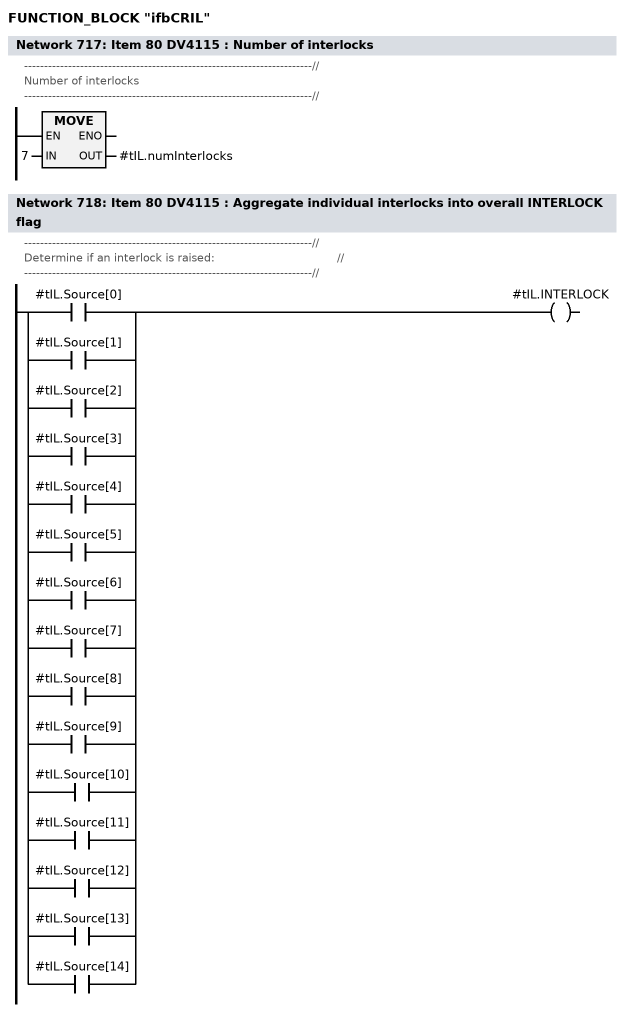
    L 7;
    T #tIL.numInterlocks;

NETWORK
TITLE = Item 80 DV4115 : Aggregate individual interlocks into overall INTERLOCK flag
    //------------------------------------------------------------------------//
    // Determine if an interlock is raised:                                   //
    //------------------------------------------------------------------------//
    O #tIL.Source[0];
    O #tIL.Source[1];
    O #tIL.Source[2];
    O #tIL.Source[3];
    O #tIL.Source[4];
    O #tIL.Source[5];
    O #tIL.Source[6];
    O #tIL.Source[7];
    O #tIL.Source[8];
    O #tIL.Source[9];
    O #tIL.Source[10];
    O #tIL.Source[11];
    O #tIL.Source[12];
    O #tIL.Source[13];
    O #tIL.Source[14];
    = #tIL.INTERLOCK;

NETWORK
TITLE = Item 80 DV4115 : Update the instance data
    //------------------------------------------------------------------------//
    // Update the instance DB with the calculated interlock flags:            //
    //------------------------------------------------------------------------//
    CALL MOVE
    {value_type := 'Variant'}
    (   IN                   := #tIL ,
        OUT                  := #p[80]
    );

NETWORK
TITLE = Item 81 DV4117 : Spray Ball 1 Valve initialise variables
    //------------------------------------------------------------------------//
    // CRITICAL INTERLOCK   CRITICAL INTERLOCK   CRITICAL INTERLOCK   CRITICA //
    // CRITICAL INTERLOCK   CRITICAL INTERLOCK   CRITICAL INTERLOCK   CRITICA //
    //                                                                        //
    // Clear the interlock flag:                                              //
    //------------------------------------------------------------------------//
    A "alwaysLow";
    = #tIL.INTERLOCK;

    //------------------------------------------------------------------------//
    // Clear all interlock values to initialise them to off:                  //
    //------------------------------------------------------------------------//
    CALL FILL_BLK
    {value_type := 'Bool', count_type := 'UInt'}
    (   IN                   := 0 ,
        COUNT                := 15 ,
        OUT                  := #tIL.Source[0]
    );


NETWORK
TITLE = Item 81 DV4117 interlock source : A RD4101 Vessel Burst Disc ALARM
    //------------------------------------------------------------------------//
    // Calculate the interlock condition:                                     //
    //------------------------------------------------------------------------//
    A idbDI1.f[16].p.read.mc.INTERLOCK;
    = #tIL.Source[0];

NETWORK
TITLE = Item 81 DV4117 interlock source : A ES4100 Vessel Emergency Stop mounted on HMI INTERLOCK
    //------------------------------------------------------------------------//
    // Calculate the interlock condition:                                     //
    //------------------------------------------------------------------------//
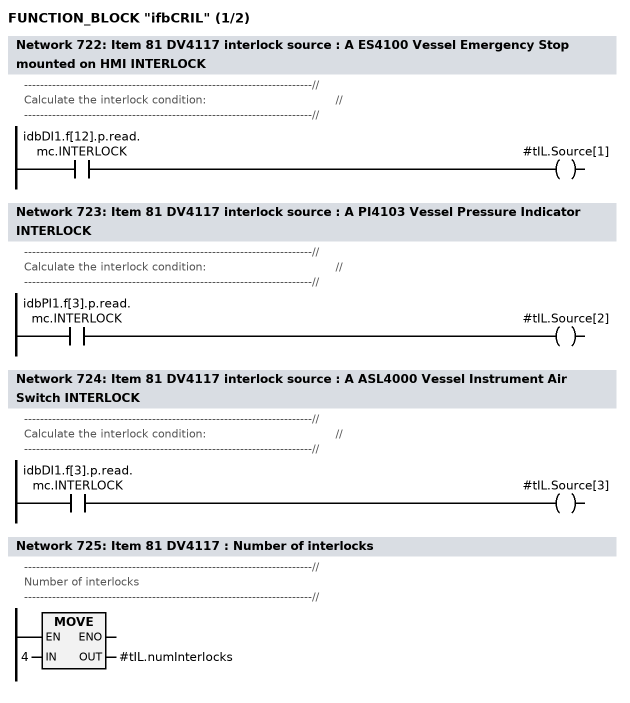
    A idbDI1.f[12].p.read.mc.INTERLOCK;
    = #tIL.Source[1];

NETWORK
TITLE = Item 81 DV4117 interlock source : A PI4103 Vessel Pressure Indicator INTERLOCK
    //------------------------------------------------------------------------//
    // Calculate the interlock condition:                                     //
    //------------------------------------------------------------------------//
    A idbPI1.f[3].p.read.mc.INTERLOCK;
    = #tIL.Source[2];

NETWORK
TITLE = Item 81 DV4117 interlock source : A ASL4000 Vessel Instrument Air Switch INTERLOCK
    //------------------------------------------------------------------------//
    // Calculate the interlock condition:                                     //
    //------------------------------------------------------------------------//
    A idbDI1.f[3].p.read.mc.INTERLOCK;
    = #tIL.Source[3];


NETWORK
TITLE = Item 81 DV4117 : Number of interlocks
    //------------------------------------------------------------------------//
    // Number of interlocks
    //------------------------------------------------------------------------//
    L 4;
    T #tIL.numInterlocks;

NETWORK
TITLE = Item 81 DV4117 : Aggregate individual interlocks into overall INTERLOCK flag
    //------------------------------------------------------------------------//
    // Determine if an interlock is raised:                                   //
    //------------------------------------------------------------------------//
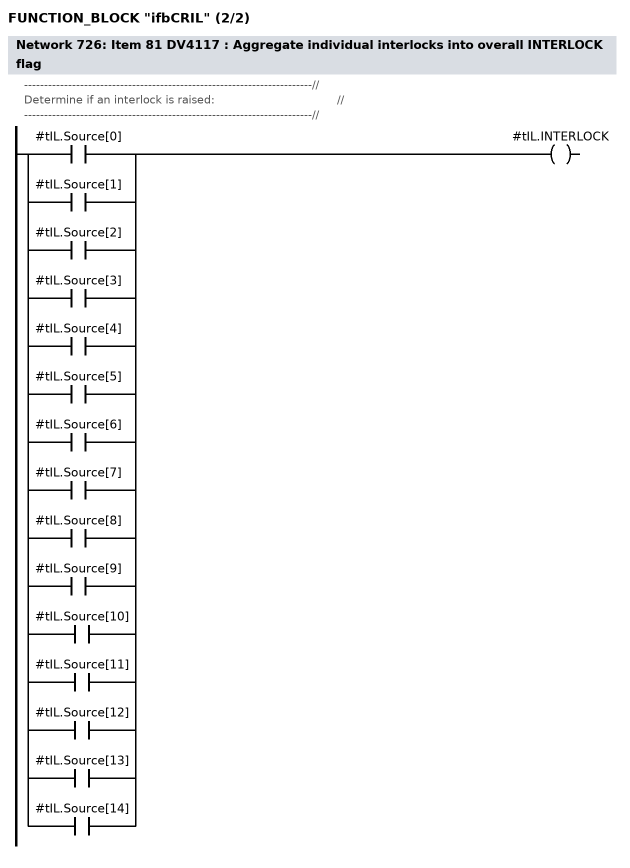
    O #tIL.Source[0];
    O #tIL.Source[1];
    O #tIL.Source[2];
    O #tIL.Source[3];
    O #tIL.Source[4];
    O #tIL.Source[5];
    O #tIL.Source[6];
    O #tIL.Source[7];
    O #tIL.Source[8];
    O #tIL.Source[9];
    O #tIL.Source[10];
    O #tIL.Source[11];
    O #tIL.Source[12];
    O #tIL.Source[13];
    O #tIL.Source[14];
    = #tIL.INTERLOCK;

NETWORK
TITLE = Item 81 DV4117 : Update the instance data
    //------------------------------------------------------------------------//
    // Update the instance DB with the calculated interlock flags:            //
    //------------------------------------------------------------------------//
    CALL MOVE
    {value_type := 'Variant'}
    (   IN                   := #tIL ,
        OUT                  := #p[81]
    );

NETWORK
TITLE = Item 82 DV4119 : Spray Ball 2 Valve initialise variables
    //------------------------------------------------------------------------//
    // CRITICAL INTERLOCK   CRITICAL INTERLOCK   CRITICAL INTERLOCK   CRITICA //
    // CRITICAL INTERLOCK   CRITICAL INTERLOCK   CRITICAL INTERLOCK   CRITICA //
    //                                                                        //
    // Clear the interlock flag:                                              //
    //------------------------------------------------------------------------//
    A "alwaysLow";
    = #tIL.INTERLOCK;

    //------------------------------------------------------------------------//
    // Clear all interlock values to initialise them to off:                  //
    //------------------------------------------------------------------------//
    CALL FILL_BLK
    {value_type := 'Bool', count_type := 'UInt'}
    (   IN                   := 0 ,
        COUNT                := 15 ,
        OUT                  := #tIL.Source[0]
    );


NETWORK
TITLE = Item 82 DV4119 interlock source : A RD4101 Vessel Burst Disc ALARM
    //------------------------------------------------------------------------//
    // Calculate the interlock condition:                                     //
    //------------------------------------------------------------------------//
    A idbDI1.f[16].p.read.mc.INTERLOCK;
    = #tIL.Source[0];

NETWORK
TITLE = Item 82 DV4119 interlock source : A ES4100 Vessel Emergency Stop mounted on HMI INTERLOCK
    //------------------------------------------------------------------------//
    // Calculate the interlock condition:                                     //
    //------------------------------------------------------------------------//
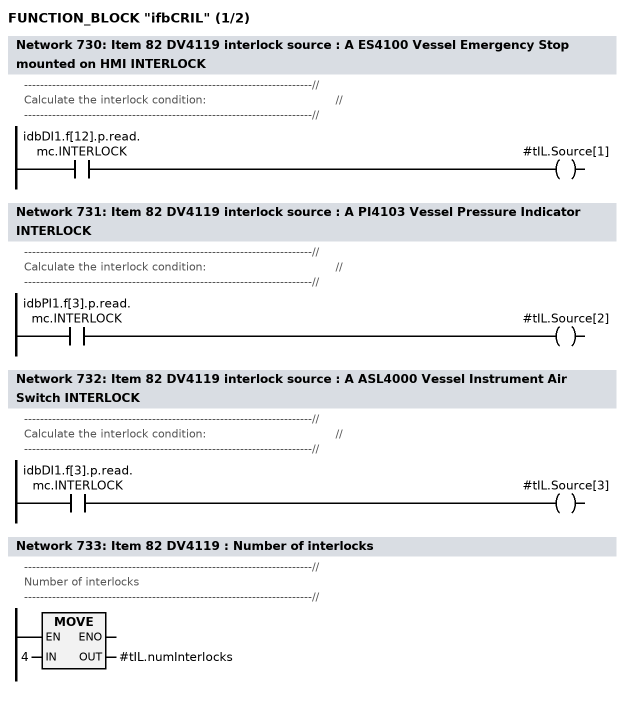
    A idbDI1.f[12].p.read.mc.INTERLOCK;
    = #tIL.Source[1];

NETWORK
TITLE = Item 82 DV4119 interlock source : A PI4103 Vessel Pressure Indicator INTERLOCK
    //------------------------------------------------------------------------//
    // Calculate the interlock condition:                                     //
    //------------------------------------------------------------------------//
    A idbPI1.f[3].p.read.mc.INTERLOCK;
    = #tIL.Source[2];

NETWORK
TITLE = Item 82 DV4119 interlock source : A ASL4000 Vessel Instrument Air Switch INTERLOCK
    //------------------------------------------------------------------------//
    // Calculate the interlock condition:                                     //
    //------------------------------------------------------------------------//
    A idbDI1.f[3].p.read.mc.INTERLOCK;
    = #tIL.Source[3];


NETWORK
TITLE = Item 82 DV4119 : Number of interlocks
    //------------------------------------------------------------------------//
    // Number of interlocks
    //------------------------------------------------------------------------//
    L 4;
    T #tIL.numInterlocks;

NETWORK
TITLE = Item 82 DV4119 : Aggregate individual interlocks into overall INTERLOCK flag
    //------------------------------------------------------------------------//
    // Determine if an interlock is raised:                                   //
    //------------------------------------------------------------------------//
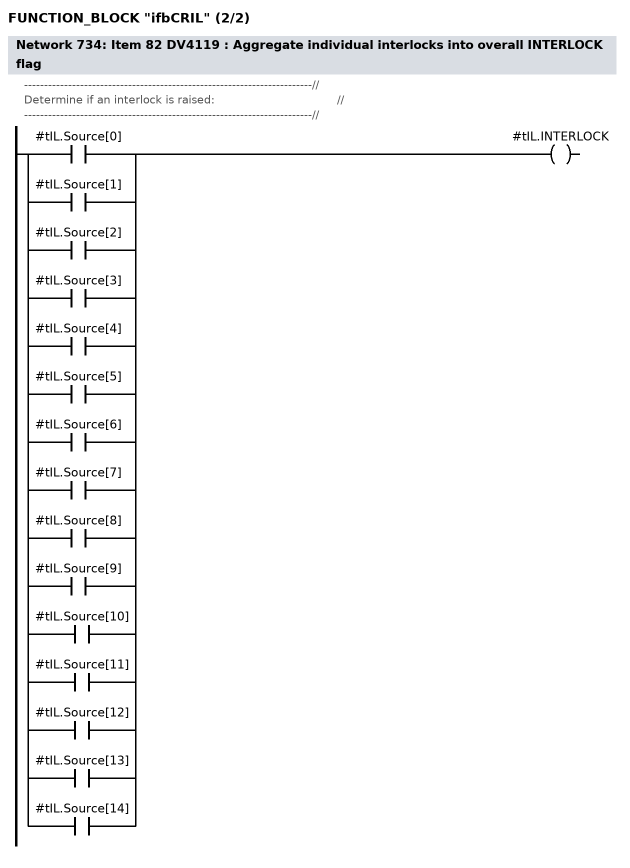
    O #tIL.Source[0];
    O #tIL.Source[1];
    O #tIL.Source[2];
    O #tIL.Source[3];
    O #tIL.Source[4];
    O #tIL.Source[5];
    O #tIL.Source[6];
    O #tIL.Source[7];
    O #tIL.Source[8];
    O #tIL.Source[9];
    O #tIL.Source[10];
    O #tIL.Source[11];
    O #tIL.Source[12];
    O #tIL.Source[13];
    O #tIL.Source[14];
    = #tIL.INTERLOCK;

NETWORK
TITLE = Item 82 DV4119 : Update the instance data
    //------------------------------------------------------------------------//
    // Update the instance DB with the calculated interlock flags:            //
    //------------------------------------------------------------------------//
    CALL MOVE
    {value_type := 'Variant'}
    (   IN                   := #tIL ,
        OUT                  := #p[82]
    );

NETWORK
TITLE = Item 83 DV4121 : Outlet Valve initialise variables
    //------------------------------------------------------------------------//
    // CRITICAL INTERLOCK   CRITICAL INTERLOCK   CRITICAL INTERLOCK   CRITICA //
    // CRITICAL INTERLOCK   CRITICAL INTERLOCK   CRITICAL INTERLOCK   CRITICA //
    //                                                                        //
    // Clear the interlock flag:                                              //
    //------------------------------------------------------------------------//
    A "alwaysLow";
    = #tIL.INTERLOCK;

    //------------------------------------------------------------------------//
    // Clear all interlock values to initialise them to off:                  //
    //------------------------------------------------------------------------//
    CALL FILL_BLK
    {value_type := 'Bool', count_type := 'UInt'}
    (   IN                   := 0 ,
        COUNT                := 15 ,
        OUT                  := #tIL.Source[0]
    );


NETWORK
TITLE = Item 83 DV4121 interlock source : A RD4101 Vessel Burst Disc ALARM
    //------------------------------------------------------------------------//
    // Calculate the interlock condition:                                     //
    //------------------------------------------------------------------------//
    A idbDI1.f[16].p.read.mc.INTERLOCK;
    = #tIL.Source[0];

NETWORK
TITLE = Item 83 DV4121 interlock source : A ES4100 Vessel Emergency Stop mounted on HMI INTERLOCK
    //------------------------------------------------------------------------//
    // Calculate the interlock condition:                                     //
    //------------------------------------------------------------------------//
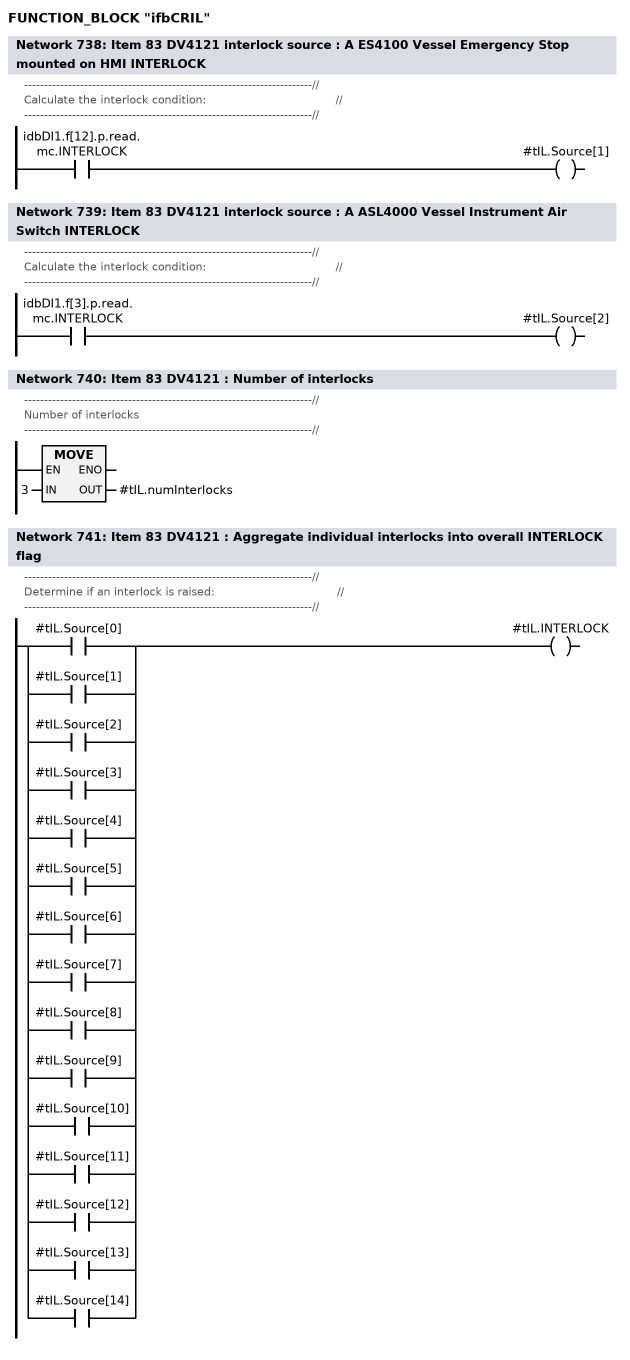
    A idbDI1.f[12].p.read.mc.INTERLOCK;
    = #tIL.Source[1];

NETWORK
TITLE = Item 83 DV4121 interlock source : A ASL4000 Vessel Instrument Air Switch INTERLOCK
    //------------------------------------------------------------------------//
    // Calculate the interlock condition:                                     //
    //------------------------------------------------------------------------//
    A idbDI1.f[3].p.read.mc.INTERLOCK;
    = #tIL.Source[2];


NETWORK
TITLE = Item 83 DV4121 : Number of interlocks
    //------------------------------------------------------------------------//
    // Number of interlocks
    //------------------------------------------------------------------------//
    L 3;
    T #tIL.numInterlocks;

NETWORK
TITLE = Item 83 DV4121 : Aggregate individual interlocks into overall INTERLOCK flag
    //------------------------------------------------------------------------//
    // Determine if an interlock is raised:                                   //
    //------------------------------------------------------------------------//
    O #tIL.Source[0];
    O #tIL.Source[1];
    O #tIL.Source[2];
    O #tIL.Source[3];
    O #tIL.Source[4];
    O #tIL.Source[5];
    O #tIL.Source[6];
    O #tIL.Source[7];
    O #tIL.Source[8];
    O #tIL.Source[9];
    O #tIL.Source[10];
    O #tIL.Source[11];
    O #tIL.Source[12];
    O #tIL.Source[13];
    O #tIL.Source[14];
    = #tIL.INTERLOCK;

NETWORK
TITLE = Item 83 DV4121 : Update the instance data
    //------------------------------------------------------------------------//
    // Update the instance DB with the calculated interlock flags:            //
    //------------------------------------------------------------------------//
    CALL MOVE
    {value_type := 'Variant'}
    (   IN                   := #tIL ,
        OUT                  := #p[83]
    );

NETWORK
TITLE = Item 84 DV4125 : Sy Transfer line Valve Matrix SMFLx initialise variables
    //------------------------------------------------------------------------//
    // CRITICAL INTERLOCK   CRITICAL INTERLOCK   CRITICAL INTERLOCK   CRITICA //
    // CRITICAL INTERLOCK   CRITICAL INTERLOCK   CRITICAL INTERLOCK   CRITICA //
    //                                                                        //
    // Clear the interlock flag:                                              //
    //------------------------------------------------------------------------//
    A "alwaysLow";
    = #tIL.INTERLOCK;

    //------------------------------------------------------------------------//
    // Clear all interlock values to initialise them to off:                  //
    //------------------------------------------------------------------------//
    CALL FILL_BLK
    {value_type := 'Bool', count_type := 'UInt'}
    (   IN                   := 0 ,
        COUNT                := 15 ,
        OUT                  := #tIL.Source[0]
    );


NETWORK
TITLE = Item 84 DV4125 interlock source : AN ZSC4111 SMFL1 to S1/BFS1 Flowpath Indicator IN   AN ZSC4113 SMFL2 to S1/BFS1 Flowpath Indicator IN
    //------------------------------------------------------------------------//
    // Calculate the interlock condition:                                     //
    //------------------------------------------------------------------------//
    AN(;
    L "idbZSC2".f[24].p.read.mc.STATE;
    L "dbCONST".BLK.ZSC2.STATE.IN;
    ==I;
    );
AN(;
    L "idbZSC2".f[25].p.read.mc.STATE;
    L "dbCONST".BLK.ZSC2.STATE.IN;
    ==I;
    );
    = #tIL.Source[0];


NETWORK
TITLE = Item 84 DV4125 : Number of interlocks
    //------------------------------------------------------------------------//
    // Number of interlocks
    //------------------------------------------------------------------------//
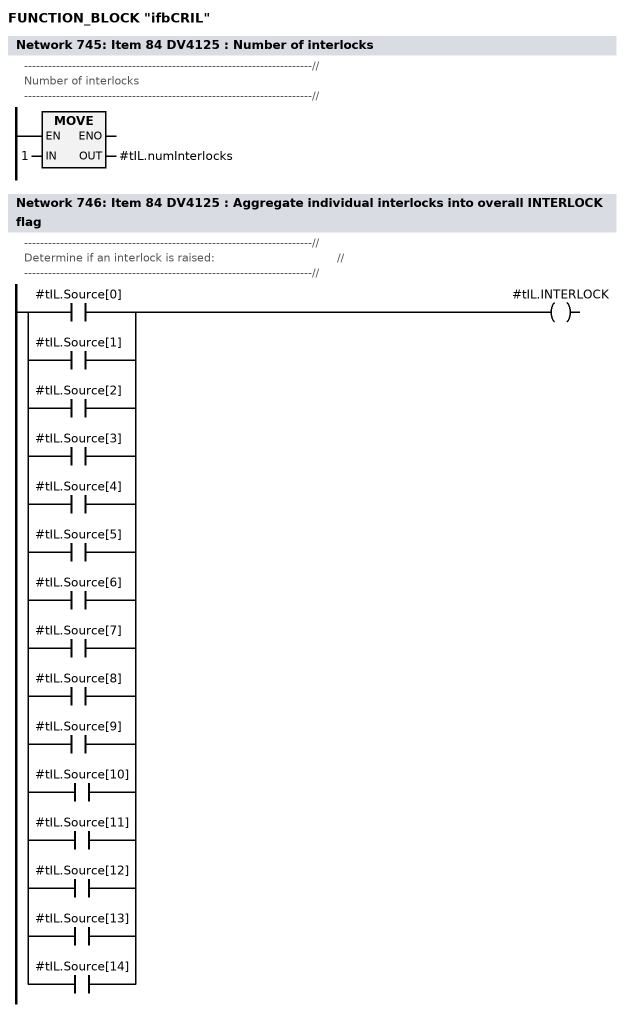
    L 1;
    T #tIL.numInterlocks;

NETWORK
TITLE = Item 84 DV4125 : Aggregate individual interlocks into overall INTERLOCK flag
    //------------------------------------------------------------------------//
    // Determine if an interlock is raised:                                   //
    //------------------------------------------------------------------------//
    O #tIL.Source[0];
    O #tIL.Source[1];
    O #tIL.Source[2];
    O #tIL.Source[3];
    O #tIL.Source[4];
    O #tIL.Source[5];
    O #tIL.Source[6];
    O #tIL.Source[7];
    O #tIL.Source[8];
    O #tIL.Source[9];
    O #tIL.Source[10];
    O #tIL.Source[11];
    O #tIL.Source[12];
    O #tIL.Source[13];
    O #tIL.Source[14];
    = #tIL.INTERLOCK;

NETWORK
TITLE = Item 84 DV4125 : Update the instance data
    //------------------------------------------------------------------------//
    // Update the instance DB with the calculated interlock flags:            //
    //------------------------------------------------------------------------//
    CALL MOVE
    {value_type := 'Variant'}
    (   IN                   := #tIL ,
        OUT                  := #p[84]
    );

NETWORK
TITLE = Item 85 DV4129 : Sy Transfer line Valve Matrix FLz initialise variables
    //------------------------------------------------------------------------//
    // CRITICAL INTERLOCK   CRITICAL INTERLOCK   CRITICAL INTERLOCK   CRITICA //
    // CRITICAL INTERLOCK   CRITICAL INTERLOCK   CRITICAL INTERLOCK   CRITICA //
    //                                                                        //
    // Clear the interlock flag:                                              //
    //------------------------------------------------------------------------//
    A "alwaysLow";
    = #tIL.INTERLOCK;

    //------------------------------------------------------------------------//
    // Clear all interlock values to initialise them to off:                  //
    //------------------------------------------------------------------------//
    CALL FILL_BLK
    {value_type := 'Bool', count_type := 'UInt'}
    (   IN                   := 0 ,
        COUNT                := 15 ,
        OUT                  := #tIL.Source[0]
    );


NETWORK
TITLE = Item 85 DV4129 interlock source : AN ZSC4115 S1 to F1P1 Flowpath Indicator IN   AN ZSC4117 S1 to F2P1 Flowpath Indicator IN
    //------------------------------------------------------------------------//
    // Calculate the interlock condition:                                     //
    //------------------------------------------------------------------------//
    AN(;
    L "idbZSC2".f[26].p.read.mc.STATE;
    L "dbCONST".BLK.ZSC2.STATE.IN;
    ==I;
    );
AN(;
    L "idbZSC2".f[27].p.read.mc.STATE;
    L "dbCONST".BLK.ZSC2.STATE.IN;
    ==I;
    );
    = #tIL.Source[0];


NETWORK
TITLE = Item 85 DV4129 : Number of interlocks
    //------------------------------------------------------------------------//
    // Number of interlocks
    //------------------------------------------------------------------------//
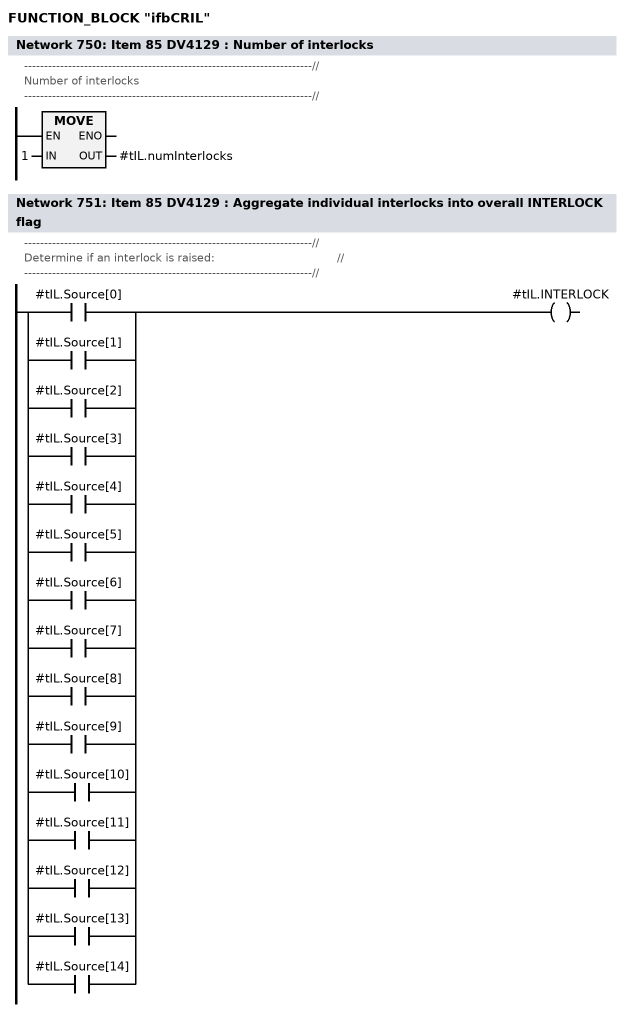
    L 1;
    T #tIL.numInterlocks;

NETWORK
TITLE = Item 85 DV4129 : Aggregate individual interlocks into overall INTERLOCK flag
    //------------------------------------------------------------------------//
    // Determine if an interlock is raised:                                   //
    //------------------------------------------------------------------------//
    O #tIL.Source[0];
    O #tIL.Source[1];
    O #tIL.Source[2];
    O #tIL.Source[3];
    O #tIL.Source[4];
    O #tIL.Source[5];
    O #tIL.Source[6];
    O #tIL.Source[7];
    O #tIL.Source[8];
    O #tIL.Source[9];
    O #tIL.Source[10];
    O #tIL.Source[11];
    O #tIL.Source[12];
    O #tIL.Source[13];
    O #tIL.Source[14];
    = #tIL.INTERLOCK;

NETWORK
TITLE = Item 85 DV4129 : Update the instance data
    //------------------------------------------------------------------------//
    // Update the instance DB with the calculated interlock flags:            //
    //------------------------------------------------------------------------//
    CALL MOVE
    {value_type := 'Variant'}
    (   IN                   := #tIL ,
        OUT                  := #p[85]
    );

NETWORK
TITLE = Item 86 HE1101 : Electric Heating Element initialise variables
    //------------------------------------------------------------------------//
    // CRITICAL INTERLOCK   CRITICAL INTERLOCK   CRITICAL INTERLOCK   CRITICA //
    // CRITICAL INTERLOCK   CRITICAL INTERLOCK   CRITICAL INTERLOCK   CRITICA //
    //                                                                        //
    // Clear the interlock flag:                                              //
    //------------------------------------------------------------------------//
    A "alwaysLow";
    = #tIL.INTERLOCK;

    //------------------------------------------------------------------------//
    // Clear all interlock values to initialise them to off:                  //
    //------------------------------------------------------------------------//
    CALL FILL_BLK
    {value_type := 'Bool', count_type := 'UInt'}
    (   IN                   := 0 ,
        COUNT                := 15 ,
        OUT                  := #tIL.Source[0]
    );


NETWORK
TITLE = Item 86 HE1101 interlock source : A RD1101 Vessel Burst Disc ALARM
    //------------------------------------------------------------------------//
    // Calculate the interlock condition:                                     //
    //------------------------------------------------------------------------//
    A idbDI1.f[13].p.read.mc.INTERLOCK;
    = #tIL.Source[0];

NETWORK
TITLE = Item 86 HE1101 interlock source : A ES1100 Vessel Emergency Stop mounted on HMI INTERLOCK
    //------------------------------------------------------------------------//
    // Calculate the interlock condition:                                     //
    //------------------------------------------------------------------------//
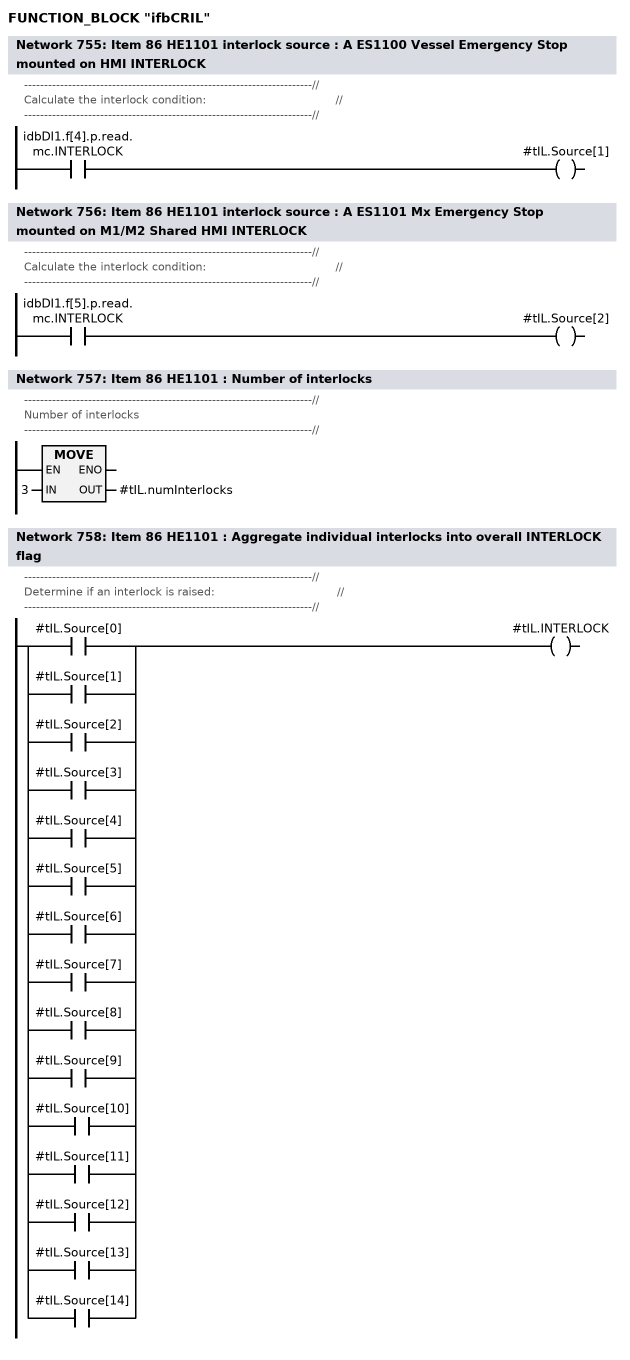
    A idbDI1.f[4].p.read.mc.INTERLOCK;
    = #tIL.Source[1];

NETWORK
TITLE = Item 86 HE1101 interlock source : A ES1101 Mx Emergency Stop mounted on M1/M2 Shared HMI INTERLOCK
    //------------------------------------------------------------------------//
    // Calculate the interlock condition:                                     //
    //------------------------------------------------------------------------//
    A idbDI1.f[5].p.read.mc.INTERLOCK;
    = #tIL.Source[2];


NETWORK
TITLE = Item 86 HE1101 : Number of interlocks
    //------------------------------------------------------------------------//
    // Number of interlocks
    //------------------------------------------------------------------------//
    L 3;
    T #tIL.numInterlocks;

NETWORK
TITLE = Item 86 HE1101 : Aggregate individual interlocks into overall INTERLOCK flag
    //------------------------------------------------------------------------//
    // Determine if an interlock is raised:                                   //
    //------------------------------------------------------------------------//
    O #tIL.Source[0];
    O #tIL.Source[1];
    O #tIL.Source[2];
    O #tIL.Source[3];
    O #tIL.Source[4];
    O #tIL.Source[5];
    O #tIL.Source[6];
    O #tIL.Source[7];
    O #tIL.Source[8];
    O #tIL.Source[9];
    O #tIL.Source[10];
    O #tIL.Source[11];
    O #tIL.Source[12];
    O #tIL.Source[13];
    O #tIL.Source[14];
    = #tIL.INTERLOCK;

NETWORK
TITLE = Item 86 HE1101 : Update the instance data
    //------------------------------------------------------------------------//
    // Update the instance DB with the calculated interlock flags:            //
    //------------------------------------------------------------------------//
    CALL MOVE
    {value_type := 'Variant'}
    (   IN                   := #tIL ,
        OUT                  := #p[86]
    );

NETWORK
TITLE = Item 87 HE2101 : Electric Heating Element initialise variables
    //------------------------------------------------------------------------//
    // CRITICAL INTERLOCK   CRITICAL INTERLOCK   CRITICAL INTERLOCK   CRITICA //
    // CRITICAL INTERLOCK   CRITICAL INTERLOCK   CRITICAL INTERLOCK   CRITICA //
    //                                                                        //
    // Clear the interlock flag:                                              //
    //------------------------------------------------------------------------//
    A "alwaysLow";
    = #tIL.INTERLOCK;

    //------------------------------------------------------------------------//
    // Clear all interlock values to initialise them to off:                  //
    //------------------------------------------------------------------------//
    CALL FILL_BLK
    {value_type := 'Bool', count_type := 'UInt'}
    (   IN                   := 0 ,
        COUNT                := 15 ,
        OUT                  := #tIL.Source[0]
    );


NETWORK
TITLE = Item 87 HE2101 interlock source : A RD2101 Vessel Burst Disc ALARM
    //------------------------------------------------------------------------//
    // Calculate the interlock condition:                                     //
    //------------------------------------------------------------------------//
    A idbDI1.f[14].p.read.mc.INTERLOCK;
    = #tIL.Source[0];

NETWORK
TITLE = Item 87 HE2101 interlock source : A ES2100 Vessel Emergency Stop mounted on HMI INTERLOCK
    //------------------------------------------------------------------------//
    // Calculate the interlock condition:                                     //
    //------------------------------------------------------------------------//
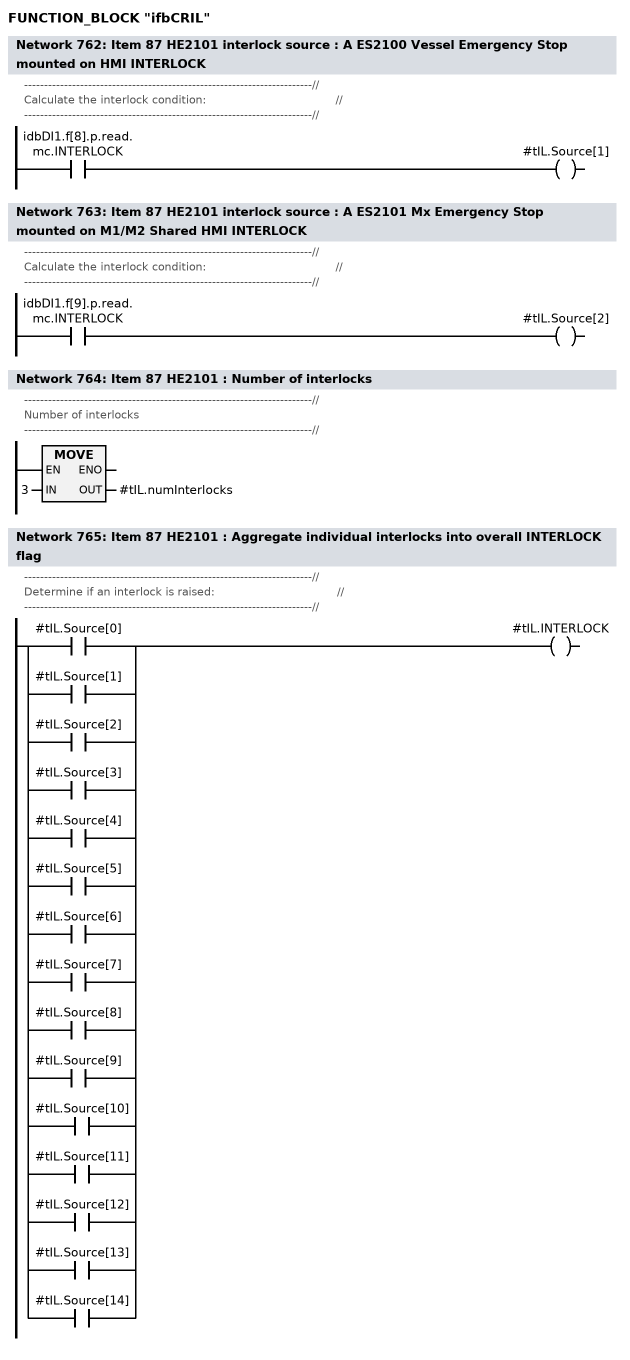
    A idbDI1.f[8].p.read.mc.INTERLOCK;
    = #tIL.Source[1];

NETWORK
TITLE = Item 87 HE2101 interlock source : A ES2101 Mx Emergency Stop mounted on M1/M2 Shared HMI INTERLOCK
    //------------------------------------------------------------------------//
    // Calculate the interlock condition:                                     //
    //------------------------------------------------------------------------//
    A idbDI1.f[9].p.read.mc.INTERLOCK;
    = #tIL.Source[2];


NETWORK
TITLE = Item 87 HE2101 : Number of interlocks
    //------------------------------------------------------------------------//
    // Number of interlocks
    //------------------------------------------------------------------------//
    L 3;
    T #tIL.numInterlocks;

NETWORK
TITLE = Item 87 HE2101 : Aggregate individual interlocks into overall INTERLOCK flag
    //------------------------------------------------------------------------//
    // Determine if an interlock is raised:                                   //
    //------------------------------------------------------------------------//
    O #tIL.Source[0];
    O #tIL.Source[1];
    O #tIL.Source[2];
    O #tIL.Source[3];
    O #tIL.Source[4];
    O #tIL.Source[5];
    O #tIL.Source[6];
    O #tIL.Source[7];
    O #tIL.Source[8];
    O #tIL.Source[9];
    O #tIL.Source[10];
    O #tIL.Source[11];
    O #tIL.Source[12];
    O #tIL.Source[13];
    O #tIL.Source[14];
    = #tIL.INTERLOCK;

NETWORK
TITLE = Item 87 HE2101 : Update the instance data
    //------------------------------------------------------------------------//
    // Update the instance DB with the calculated interlock flags:            //
    //------------------------------------------------------------------------//
    CALL MOVE
    {value_type := 'Variant'}
    (   IN                   := #tIL ,
        OUT                  := #p[87]
    );

NETWORK
TITLE = Item 88 HE3101 : Electric Heating Element initialise variables
    //------------------------------------------------------------------------//
    // CRITICAL INTERLOCK   CRITICAL INTERLOCK   CRITICAL INTERLOCK   CRITICA //
    // CRITICAL INTERLOCK   CRITICAL INTERLOCK   CRITICAL INTERLOCK   CRITICA //
    //                                                                        //
    // Clear the interlock flag:                                              //
    //------------------------------------------------------------------------//
    A "alwaysLow";
    = #tIL.INTERLOCK;

    //------------------------------------------------------------------------//
    // Clear all interlock values to initialise them to off:                  //
    //------------------------------------------------------------------------//
    CALL FILL_BLK
    {value_type := 'Bool', count_type := 'UInt'}
    (   IN                   := 0 ,
        COUNT                := 15 ,
        OUT                  := #tIL.Source[0]
    );


NETWORK
TITLE = Item 88 HE3101 interlock source : A RD3101 Vessel Burst Disc ALARM
    //------------------------------------------------------------------------//
    // Calculate the interlock condition:                                     //
    //------------------------------------------------------------------------//
    A idbDI1.f[15].p.read.mc.INTERLOCK;
    = #tIL.Source[0];

NETWORK
TITLE = Item 88 HE3101 interlock source : A ES3100 Vessel Emergency Stop mounted on HMI INTERLOCK
    //------------------------------------------------------------------------//
    // Calculate the interlock condition:                                     //
    //------------------------------------------------------------------------//
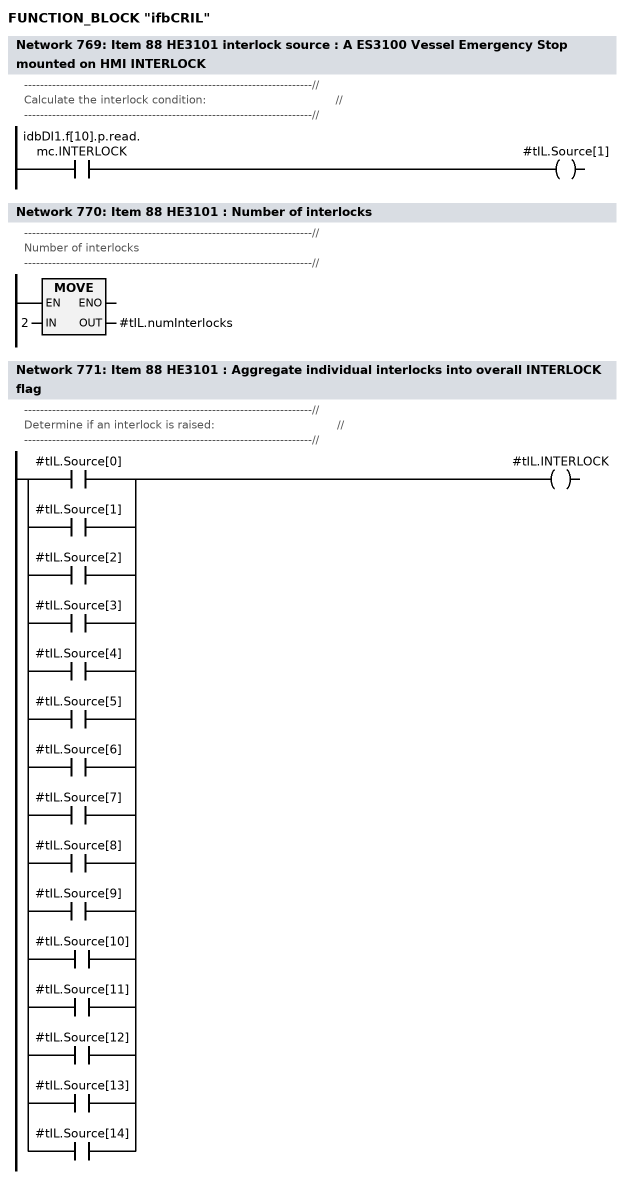
    A idbDI1.f[10].p.read.mc.INTERLOCK;
    = #tIL.Source[1];


NETWORK
TITLE = Item 88 HE3101 : Number of interlocks
    //------------------------------------------------------------------------//
    // Number of interlocks
    //------------------------------------------------------------------------//
    L 2;
    T #tIL.numInterlocks;

NETWORK
TITLE = Item 88 HE3101 : Aggregate individual interlocks into overall INTERLOCK flag
    //------------------------------------------------------------------------//
    // Determine if an interlock is raised:                                   //
    //------------------------------------------------------------------------//
    O #tIL.Source[0];
    O #tIL.Source[1];
    O #tIL.Source[2];
    O #tIL.Source[3];
    O #tIL.Source[4];
    O #tIL.Source[5];
    O #tIL.Source[6];
    O #tIL.Source[7];
    O #tIL.Source[8];
    O #tIL.Source[9];
    O #tIL.Source[10];
    O #tIL.Source[11];
    O #tIL.Source[12];
    O #tIL.Source[13];
    O #tIL.Source[14];
    = #tIL.INTERLOCK;

NETWORK
TITLE = Item 88 HE3101 : Update the instance data
    //------------------------------------------------------------------------//
    // Update the instance DB with the calculated interlock flags:            //
    //------------------------------------------------------------------------//
    CALL MOVE
    {value_type := 'Variant'}
    (   IN                   := #tIL ,
        OUT                  := #p[88]
    );

NETWORK
TITLE = Item 89 HE4101 : Electric Heating Element initialise variables
    //------------------------------------------------------------------------//
    // CRITICAL INTERLOCK   CRITICAL INTERLOCK   CRITICAL INTERLOCK   CRITICA //
    // CRITICAL INTERLOCK   CRITICAL INTERLOCK   CRITICAL INTERLOCK   CRITICA //
    //                                                                        //
    // Clear the interlock flag:                                              //
    //------------------------------------------------------------------------//
    A "alwaysLow";
    = #tIL.INTERLOCK;

    //------------------------------------------------------------------------//
    // Clear all interlock values to initialise them to off:                  //
    //------------------------------------------------------------------------//
    CALL FILL_BLK
    {value_type := 'Bool', count_type := 'UInt'}
    (   IN                   := 0 ,
        COUNT                := 15 ,
        OUT                  := #tIL.Source[0]
    );


NETWORK
TITLE = Item 89 HE4101 interlock source : A RD4101 Vessel Burst Disc ALARM
    //------------------------------------------------------------------------//
    // Calculate the interlock condition:                                     //
    //------------------------------------------------------------------------//
    A idbDI1.f[16].p.read.mc.INTERLOCK;
    = #tIL.Source[0];

NETWORK
TITLE = Item 89 HE4101 interlock source : A ES4100 Vessel Emergency Stop mounted on HMI INTERLOCK
    //------------------------------------------------------------------------//
    // Calculate the interlock condition:                                     //
    //------------------------------------------------------------------------//
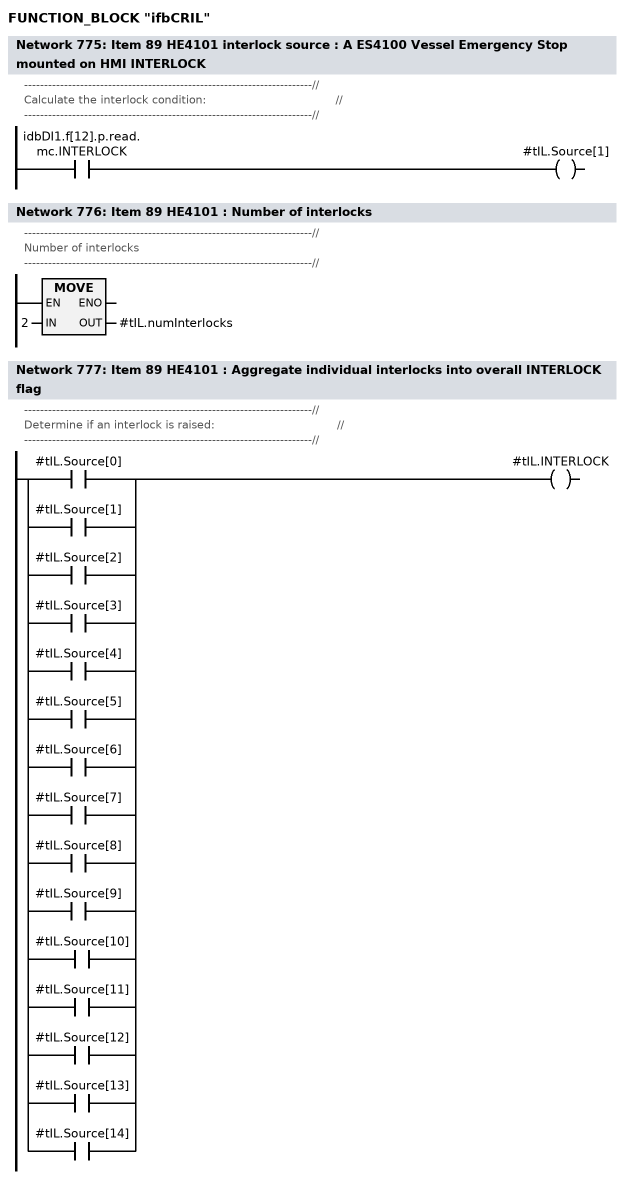
    A idbDI1.f[12].p.read.mc.INTERLOCK;
    = #tIL.Source[1];


NETWORK
TITLE = Item 89 HE4101 : Number of interlocks
    //------------------------------------------------------------------------//
    // Number of interlocks
    //------------------------------------------------------------------------//
    L 2;
    T #tIL.numInterlocks;

NETWORK
TITLE = Item 89 HE4101 : Aggregate individual interlocks into overall INTERLOCK flag
    //------------------------------------------------------------------------//
    // Determine if an interlock is raised:                                   //
    //------------------------------------------------------------------------//
    O #tIL.Source[0];
    O #tIL.Source[1];
    O #tIL.Source[2];
    O #tIL.Source[3];
    O #tIL.Source[4];
    O #tIL.Source[5];
    O #tIL.Source[6];
    O #tIL.Source[7];
    O #tIL.Source[8];
    O #tIL.Source[9];
    O #tIL.Source[10];
    O #tIL.Source[11];
    O #tIL.Source[12];
    O #tIL.Source[13];
    O #tIL.Source[14];
    = #tIL.INTERLOCK;

NETWORK
TITLE = Item 89 HE4101 : Update the instance data
    //------------------------------------------------------------------------//
    // Update the instance DB with the calculated interlock flags:            //
    //------------------------------------------------------------------------//
    CALL MOVE
    {value_type := 'Variant'}
    (   IN                   := #tIL ,
        OUT                  := #p[89]
    );

NETWORK
TITLE = Item 90 PC1103 : Pressure Control initialise variables
    //------------------------------------------------------------------------//
    // CRITICAL INTERLOCK   CRITICAL INTERLOCK   CRITICAL INTERLOCK   CRITICA //
    // CRITICAL INTERLOCK   CRITICAL INTERLOCK   CRITICAL INTERLOCK   CRITICA //
    //                                                                        //
    // Clear the interlock flag:                                              //
    //------------------------------------------------------------------------//
    A "alwaysLow";
    = #tIL.INTERLOCK;

    //------------------------------------------------------------------------//
    // Clear all interlock values to initialise them to off:                  //
    //------------------------------------------------------------------------//
    CALL FILL_BLK
    {value_type := 'Bool', count_type := 'UInt'}
    (   IN                   := 0 ,
        COUNT                := 15 ,
        OUT                  := #tIL.Source[0]
    );


NETWORK
TITLE = Item 90 PC1103 interlock source : A RD1101 Vessel Burst Disc ALARM
    //------------------------------------------------------------------------//
    // Calculate the interlock condition:                                     //
    //------------------------------------------------------------------------//
    A idbDI1.f[13].p.read.mc.INTERLOCK;
    = #tIL.Source[0];

NETWORK
TITLE = Item 90 PC1103 interlock source : A ES1100 Vessel Emergency Stop mounted on HMI INTERLOCK
    //------------------------------------------------------------------------//
    // Calculate the interlock condition:                                     //
    //------------------------------------------------------------------------//
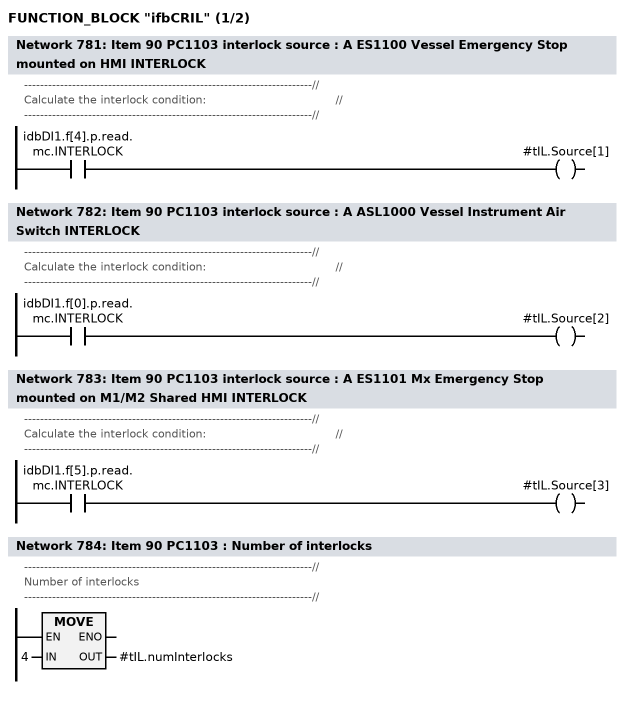
    A idbDI1.f[4].p.read.mc.INTERLOCK;
    = #tIL.Source[1];

NETWORK
TITLE = Item 90 PC1103 interlock source : A ASL1000 Vessel Instrument Air Switch INTERLOCK
    //------------------------------------------------------------------------//
    // Calculate the interlock condition:                                     //
    //------------------------------------------------------------------------//
    A idbDI1.f[0].p.read.mc.INTERLOCK;
    = #tIL.Source[2];

NETWORK
TITLE = Item 90 PC1103 interlock source : A ES1101 Mx Emergency Stop mounted on M1/M2 Shared HMI INTERLOCK
    //------------------------------------------------------------------------//
    // Calculate the interlock condition:                                     //
    //------------------------------------------------------------------------//
    A idbDI1.f[5].p.read.mc.INTERLOCK;
    = #tIL.Source[3];


NETWORK
TITLE = Item 90 PC1103 : Number of interlocks
    //------------------------------------------------------------------------//
    // Number of interlocks
    //------------------------------------------------------------------------//
    L 4;
    T #tIL.numInterlocks;

NETWORK
TITLE = Item 90 PC1103 : Aggregate individual interlocks into overall INTERLOCK flag
    //------------------------------------------------------------------------//
    // Determine if an interlock is raised:                                   //
    //------------------------------------------------------------------------//
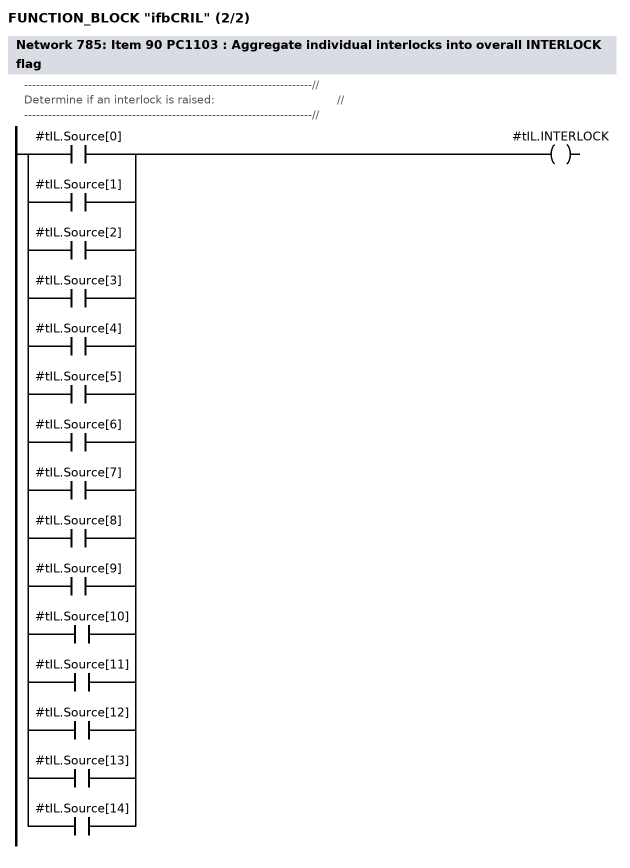
    O #tIL.Source[0];
    O #tIL.Source[1];
    O #tIL.Source[2];
    O #tIL.Source[3];
    O #tIL.Source[4];
    O #tIL.Source[5];
    O #tIL.Source[6];
    O #tIL.Source[7];
    O #tIL.Source[8];
    O #tIL.Source[9];
    O #tIL.Source[10];
    O #tIL.Source[11];
    O #tIL.Source[12];
    O #tIL.Source[13];
    O #tIL.Source[14];
    = #tIL.INTERLOCK;

NETWORK
TITLE = Item 90 PC1103 : Update the instance data
    //------------------------------------------------------------------------//
    // Update the instance DB with the calculated interlock flags:            //
    //------------------------------------------------------------------------//
    CALL MOVE
    {value_type := 'Variant'}
    (   IN                   := #tIL ,
        OUT                  := #p[90]
    );

NETWORK
TITLE = Item 91 PC2103 : Pressure Control initialise variables
    //------------------------------------------------------------------------//
    // CRITICAL INTERLOCK   CRITICAL INTERLOCK   CRITICAL INTERLOCK   CRITICA //
    // CRITICAL INTERLOCK   CRITICAL INTERLOCK   CRITICAL INTERLOCK   CRITICA //
    //                                                                        //
    // Clear the interlock flag:                                              //
    //------------------------------------------------------------------------//
    A "alwaysLow";
    = #tIL.INTERLOCK;

    //------------------------------------------------------------------------//
    // Clear all interlock values to initialise them to off:                  //
    //------------------------------------------------------------------------//
    CALL FILL_BLK
    {value_type := 'Bool', count_type := 'UInt'}
    (   IN                   := 0 ,
        COUNT                := 15 ,
        OUT                  := #tIL.Source[0]
    );


NETWORK
TITLE = Item 91 PC2103 interlock source : A RD2101 Vessel Burst Disc ALARM
    //------------------------------------------------------------------------//
    // Calculate the interlock condition:                                     //
    //------------------------------------------------------------------------//
    A idbDI1.f[14].p.read.mc.INTERLOCK;
    = #tIL.Source[0];

NETWORK
TITLE = Item 91 PC2103 interlock source : A ES2100 Vessel Emergency Stop mounted on HMI INTERLOCK
    //------------------------------------------------------------------------//
    // Calculate the interlock condition:                                     //
    //------------------------------------------------------------------------//
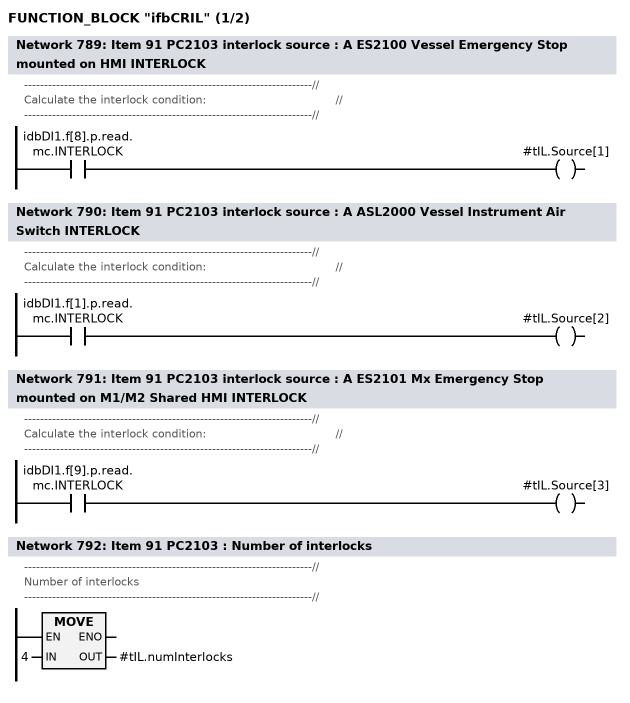
    A idbDI1.f[8].p.read.mc.INTERLOCK;
    = #tIL.Source[1];

NETWORK
TITLE = Item 91 PC2103 interlock source : A ASL2000 Vessel Instrument Air Switch INTERLOCK
    //------------------------------------------------------------------------//
    // Calculate the interlock condition:                                     //
    //------------------------------------------------------------------------//
    A idbDI1.f[1].p.read.mc.INTERLOCK;
    = #tIL.Source[2];

NETWORK
TITLE = Item 91 PC2103 interlock source : A ES2101 Mx Emergency Stop mounted on M1/M2 Shared HMI INTERLOCK
    //------------------------------------------------------------------------//
    // Calculate the interlock condition:                                     //
    //------------------------------------------------------------------------//
    A idbDI1.f[9].p.read.mc.INTERLOCK;
    = #tIL.Source[3];


NETWORK
TITLE = Item 91 PC2103 : Number of interlocks
    //------------------------------------------------------------------------//
    // Number of interlocks
    //------------------------------------------------------------------------//
    L 4;
    T #tIL.numInterlocks;

NETWORK
TITLE = Item 91 PC2103 : Aggregate individual interlocks into overall INTERLOCK flag
    //------------------------------------------------------------------------//
    // Determine if an interlock is raised:                                   //
    //------------------------------------------------------------------------//
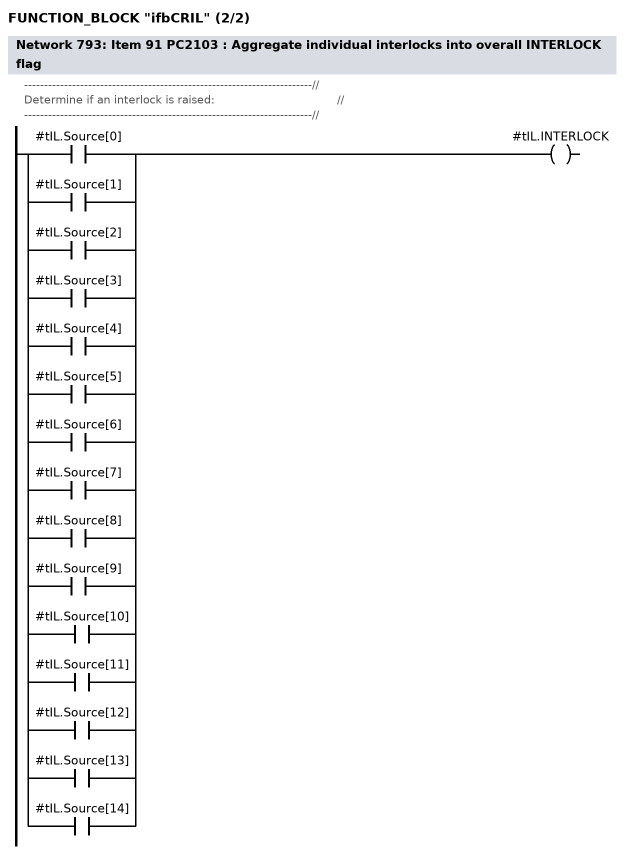
    O #tIL.Source[0];
    O #tIL.Source[1];
    O #tIL.Source[2];
    O #tIL.Source[3];
    O #tIL.Source[4];
    O #tIL.Source[5];
    O #tIL.Source[6];
    O #tIL.Source[7];
    O #tIL.Source[8];
    O #tIL.Source[9];
    O #tIL.Source[10];
    O #tIL.Source[11];
    O #tIL.Source[12];
    O #tIL.Source[13];
    O #tIL.Source[14];
    = #tIL.INTERLOCK;

NETWORK
TITLE = Item 91 PC2103 : Update the instance data
    //------------------------------------------------------------------------//
    // Update the instance DB with the calculated interlock flags:            //
    //------------------------------------------------------------------------//
    CALL MOVE
    {value_type := 'Variant'}
    (   IN                   := #tIL ,
        OUT                  := #p[91]
    );

NETWORK
TITLE = Item 92 PC3103 : Pressure Control initialise variables
    //------------------------------------------------------------------------//
    // CRITICAL INTERLOCK   CRITICAL INTERLOCK   CRITICAL INTERLOCK   CRITICA //
    // CRITICAL INTERLOCK   CRITICAL INTERLOCK   CRITICAL INTERLOCK   CRITICA //
    //                                                                        //
    // Clear the interlock flag:                                              //
    //------------------------------------------------------------------------//
    A "alwaysLow";
    = #tIL.INTERLOCK;

    //------------------------------------------------------------------------//
    // Clear all interlock values to initialise them to off:                  //
    //------------------------------------------------------------------------//
    CALL FILL_BLK
    {value_type := 'Bool', count_type := 'UInt'}
    (   IN                   := 0 ,
        COUNT                := 15 ,
        OUT                  := #tIL.Source[0]
    );


NETWORK
TITLE = Item 92 PC3103 interlock source : A RD3101 Vessel Burst Disc ALARM
    //------------------------------------------------------------------------//
    // Calculate the interlock condition:                                     //
    //------------------------------------------------------------------------//
    A idbDI1.f[15].p.read.mc.INTERLOCK;
    = #tIL.Source[0];

NETWORK
TITLE = Item 92 PC3103 interlock source : A ES3100 Vessel Emergency Stop mounted on HMI INTERLOCK
    //------------------------------------------------------------------------//
    // Calculate the interlock condition:                                     //
    //------------------------------------------------------------------------//
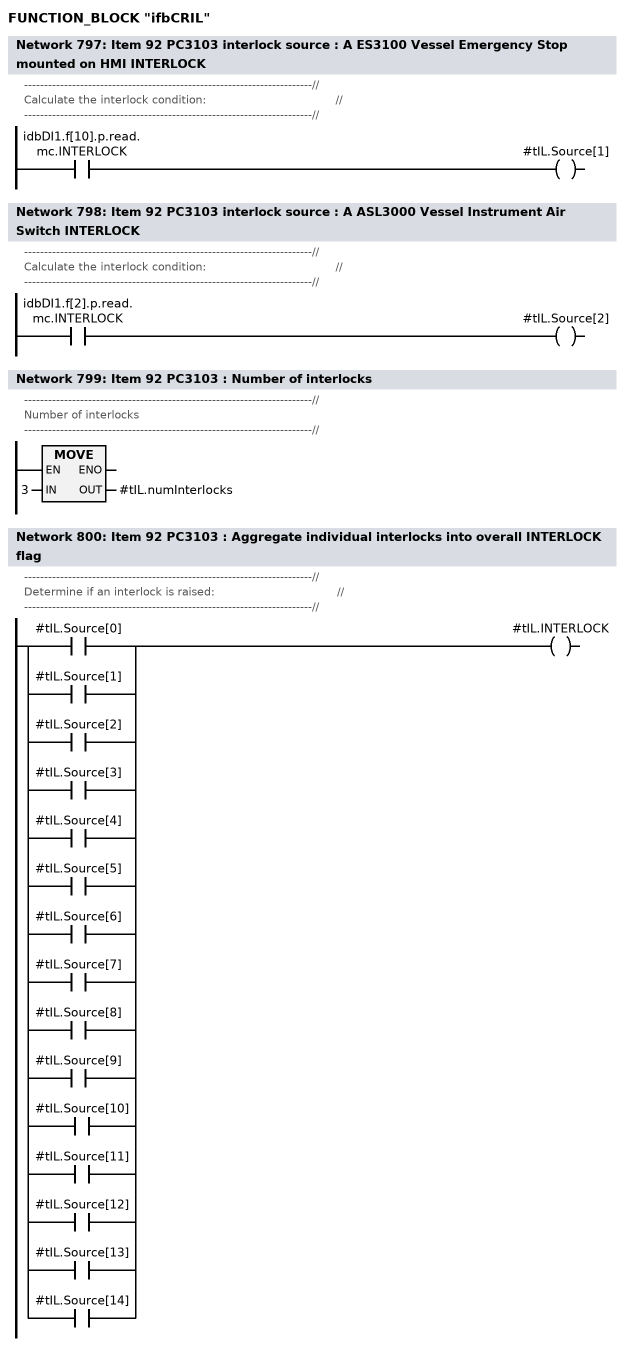
    A idbDI1.f[10].p.read.mc.INTERLOCK;
    = #tIL.Source[1];

NETWORK
TITLE = Item 92 PC3103 interlock source : A ASL3000 Vessel Instrument Air Switch INTERLOCK
    //------------------------------------------------------------------------//
    // Calculate the interlock condition:                                     //
    //------------------------------------------------------------------------//
    A idbDI1.f[2].p.read.mc.INTERLOCK;
    = #tIL.Source[2];


NETWORK
TITLE = Item 92 PC3103 : Number of interlocks
    //------------------------------------------------------------------------//
    // Number of interlocks
    //------------------------------------------------------------------------//
    L 3;
    T #tIL.numInterlocks;

NETWORK
TITLE = Item 92 PC3103 : Aggregate individual interlocks into overall INTERLOCK flag
    //------------------------------------------------------------------------//
    // Determine if an interlock is raised:                                   //
    //------------------------------------------------------------------------//
    O #tIL.Source[0];
    O #tIL.Source[1];
    O #tIL.Source[2];
    O #tIL.Source[3];
    O #tIL.Source[4];
    O #tIL.Source[5];
    O #tIL.Source[6];
    O #tIL.Source[7];
    O #tIL.Source[8];
    O #tIL.Source[9];
    O #tIL.Source[10];
    O #tIL.Source[11];
    O #tIL.Source[12];
    O #tIL.Source[13];
    O #tIL.Source[14];
    = #tIL.INTERLOCK;

NETWORK
TITLE = Item 92 PC3103 : Update the instance data
    //------------------------------------------------------------------------//
    // Update the instance DB with the calculated interlock flags:            //
    //------------------------------------------------------------------------//
    CALL MOVE
    {value_type := 'Variant'}
    (   IN                   := #tIL ,
        OUT                  := #p[92]
    );

NETWORK
TITLE = Item 93 PC4103 : Pressure Control initialise variables
    //------------------------------------------------------------------------//
    // CRITICAL INTERLOCK   CRITICAL INTERLOCK   CRITICAL INTERLOCK   CRITICA //
    // CRITICAL INTERLOCK   CRITICAL INTERLOCK   CRITICAL INTERLOCK   CRITICA //
    //                                                                        //
    // Clear the interlock flag:                                              //
    //------------------------------------------------------------------------//
    A "alwaysLow";
    = #tIL.INTERLOCK;

    //------------------------------------------------------------------------//
    // Clear all interlock values to initialise them to off:                  //
    //------------------------------------------------------------------------//
    CALL FILL_BLK
    {value_type := 'Bool', count_type := 'UInt'}
    (   IN                   := 0 ,
        COUNT                := 15 ,
        OUT                  := #tIL.Source[0]
    );


NETWORK
TITLE = Item 93 PC4103 interlock source : A RD4101 Vessel Burst Disc ALARM
    //------------------------------------------------------------------------//
    // Calculate the interlock condition:                                     //
    //------------------------------------------------------------------------//
    A idbDI1.f[16].p.read.mc.INTERLOCK;
    = #tIL.Source[0];

NETWORK
TITLE = Item 93 PC4103 interlock source : A ES4100 Vessel Emergency Stop mounted on HMI INTERLOCK
    //------------------------------------------------------------------------//
    // Calculate the interlock condition:                                     //
    //------------------------------------------------------------------------//
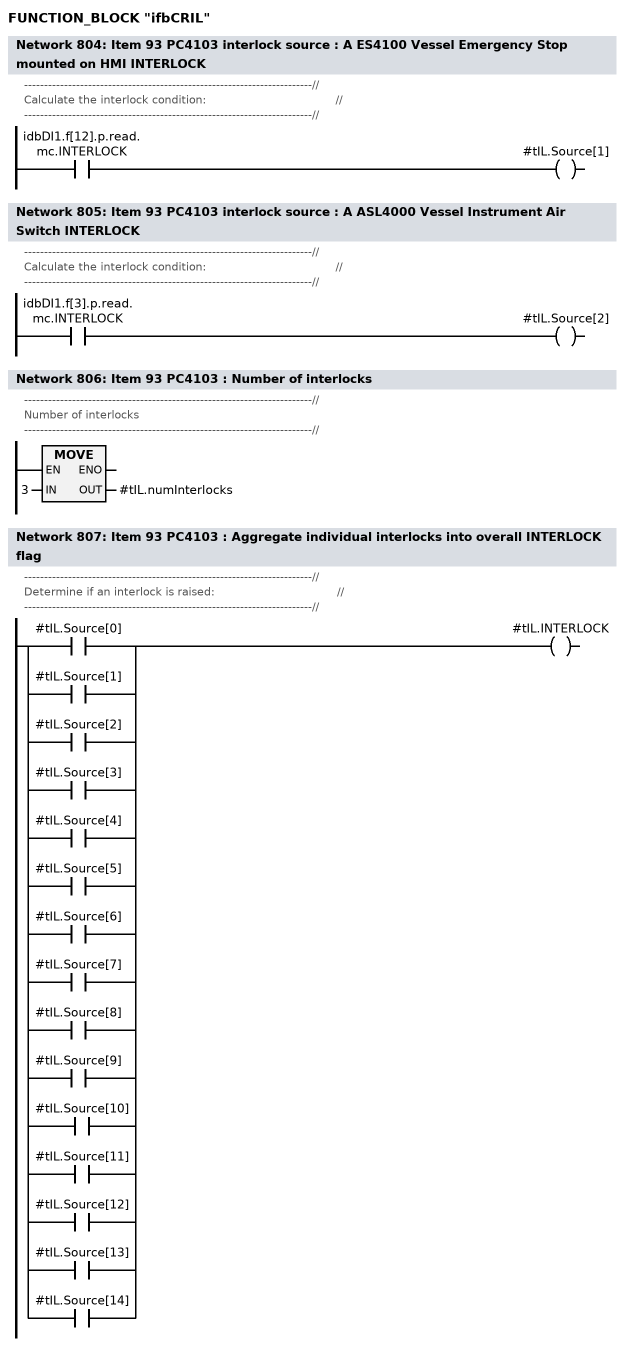
    A idbDI1.f[12].p.read.mc.INTERLOCK;
    = #tIL.Source[1];

NETWORK
TITLE = Item 93 PC4103 interlock source : A ASL4000 Vessel Instrument Air Switch INTERLOCK
    //------------------------------------------------------------------------//
    // Calculate the interlock condition:                                     //
    //------------------------------------------------------------------------//
    A idbDI1.f[3].p.read.mc.INTERLOCK;
    = #tIL.Source[2];


NETWORK
TITLE = Item 93 PC4103 : Number of interlocks
    //------------------------------------------------------------------------//
    // Number of interlocks
    //------------------------------------------------------------------------//
    L 3;
    T #tIL.numInterlocks;

NETWORK
TITLE = Item 93 PC4103 : Aggregate individual interlocks into overall INTERLOCK flag
    //------------------------------------------------------------------------//
    // Determine if an interlock is raised:                                   //
    //------------------------------------------------------------------------//
    O #tIL.Source[0];
    O #tIL.Source[1];
    O #tIL.Source[2];
    O #tIL.Source[3];
    O #tIL.Source[4];
    O #tIL.Source[5];
    O #tIL.Source[6];
    O #tIL.Source[7];
    O #tIL.Source[8];
    O #tIL.Source[9];
    O #tIL.Source[10];
    O #tIL.Source[11];
    O #tIL.Source[12];
    O #tIL.Source[13];
    O #tIL.Source[14];
    = #tIL.INTERLOCK;

NETWORK
TITLE = Item 93 PC4103 : Update the instance data
    //------------------------------------------------------------------------//
    // Update the instance DB with the calculated interlock flags:            //
    //------------------------------------------------------------------------//
    CALL MOVE
    {value_type := 'Variant'}
    (   IN                   := #tIL ,
        OUT                  := #p[93]
    );

NETWORK
TITLE = Item 94 TC1109 : MMFLx Inline Heat Exchanger Temperature Control initialise variables
    //------------------------------------------------------------------------//
    // CRITICAL INTERLOCK   CRITICAL INTERLOCK   CRITICAL INTERLOCK   CRITICA //
    // CRITICAL INTERLOCK   CRITICAL INTERLOCK   CRITICAL INTERLOCK   CRITICA //
    //                                                                        //
    // Clear the interlock flag:                                              //
    //------------------------------------------------------------------------//
    A "alwaysLow";
    = #tIL.INTERLOCK;

    //------------------------------------------------------------------------//
    // Clear all interlock values to initialise them to off:                  //
    //------------------------------------------------------------------------//
    CALL FILL_BLK
    {value_type := 'Bool', count_type := 'UInt'}
    (   IN                   := 0 ,
        COUNT                := 15 ,
        OUT                  := #tIL.Source[0]
    );


NETWORK
TITLE = Item 94 TC1109 interlock source : A RD1101 Vessel Burst Disc ALARM
    //------------------------------------------------------------------------//
    // Calculate the interlock condition:                                     //
    //------------------------------------------------------------------------//
    A idbDI1.f[13].p.read.mc.INTERLOCK;
    = #tIL.Source[0];

NETWORK
TITLE = Item 94 TC1109 interlock source : A ES1100 Vessel Emergency Stop mounted on HMI INTERLOCK
    //------------------------------------------------------------------------//
    // Calculate the interlock condition:                                     //
    //------------------------------------------------------------------------//
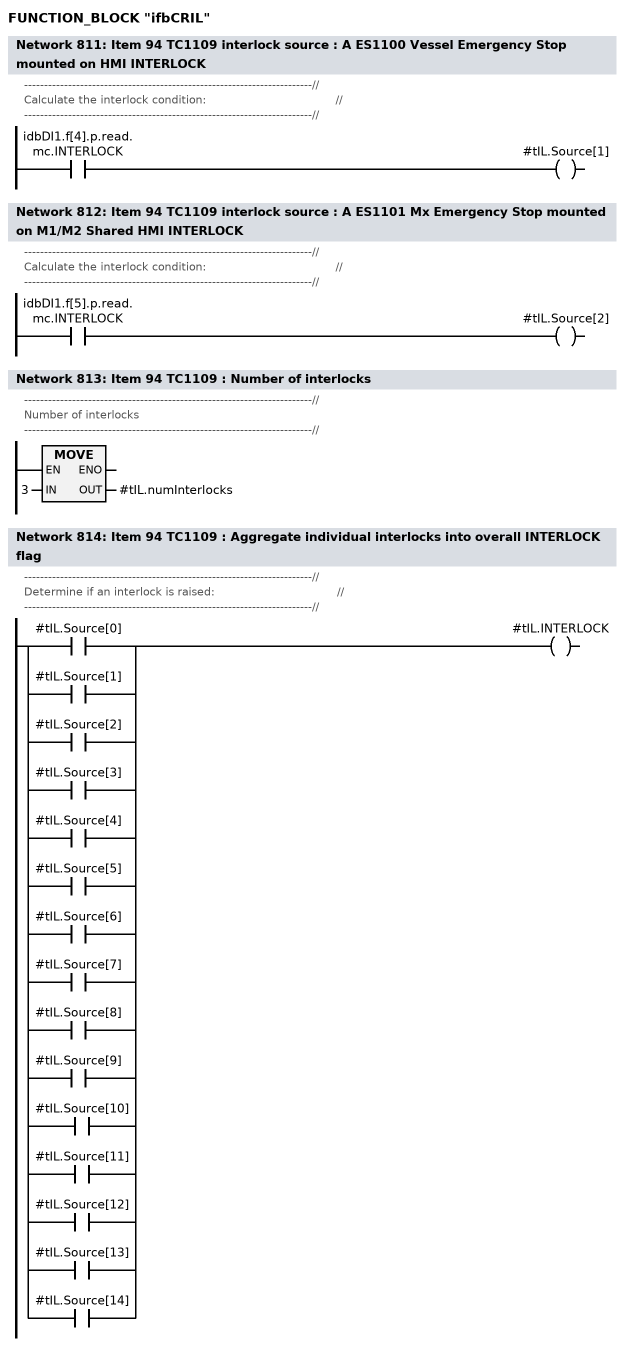
    A idbDI1.f[4].p.read.mc.INTERLOCK;
    = #tIL.Source[1];

NETWORK
TITLE = Item 94 TC1109 interlock source : A ES1101 Mx Emergency Stop mounted on M1/M2 Shared HMI INTERLOCK
    //------------------------------------------------------------------------//
    // Calculate the interlock condition:                                     //
    //------------------------------------------------------------------------//
    A idbDI1.f[5].p.read.mc.INTERLOCK;
    = #tIL.Source[2];


NETWORK
TITLE = Item 94 TC1109 : Number of interlocks
    //------------------------------------------------------------------------//
    // Number of interlocks
    //------------------------------------------------------------------------//
    L 3;
    T #tIL.numInterlocks;

NETWORK
TITLE = Item 94 TC1109 : Aggregate individual interlocks into overall INTERLOCK flag
    //------------------------------------------------------------------------//
    // Determine if an interlock is raised:                                   //
    //------------------------------------------------------------------------//
    O #tIL.Source[0];
    O #tIL.Source[1];
    O #tIL.Source[2];
    O #tIL.Source[3];
    O #tIL.Source[4];
    O #tIL.Source[5];
    O #tIL.Source[6];
    O #tIL.Source[7];
    O #tIL.Source[8];
    O #tIL.Source[9];
    O #tIL.Source[10];
    O #tIL.Source[11];
    O #tIL.Source[12];
    O #tIL.Source[13];
    O #tIL.Source[14];
    = #tIL.INTERLOCK;

NETWORK
TITLE = Item 94 TC1109 : Update the instance data
    //------------------------------------------------------------------------//
    // Update the instance DB with the calculated interlock flags:            //
    //------------------------------------------------------------------------//
    CALL MOVE
    {value_type := 'Variant'}
    (   IN                   := #tIL ,
        OUT                  := #p[94]
    );

NETWORK
TITLE = Item 95 TC2109 : MMFLx Inline Heat Exchanger Temperature Control initialise variables
    //------------------------------------------------------------------------//
    // CRITICAL INTERLOCK   CRITICAL INTERLOCK   CRITICAL INTERLOCK   CRITICA //
    // CRITICAL INTERLOCK   CRITICAL INTERLOCK   CRITICAL INTERLOCK   CRITICA //
    //                                                                        //
    // Clear the interlock flag:                                              //
    //------------------------------------------------------------------------//
    A "alwaysLow";
    = #tIL.INTERLOCK;

    //------------------------------------------------------------------------//
    // Clear all interlock values to initialise them to off:                  //
    //------------------------------------------------------------------------//
    CALL FILL_BLK
    {value_type := 'Bool', count_type := 'UInt'}
    (   IN                   := 0 ,
        COUNT                := 15 ,
        OUT                  := #tIL.Source[0]
    );


NETWORK
TITLE = Item 95 TC2109 interlock source : A RD2101 Vessel Burst Disc ALARM
    //------------------------------------------------------------------------//
    // Calculate the interlock condition:                                     //
    //------------------------------------------------------------------------//
    A idbDI1.f[14].p.read.mc.INTERLOCK;
    = #tIL.Source[0];

NETWORK
TITLE = Item 95 TC2109 interlock source : A ES2100 Vessel Emergency Stop mounted on HMI INTERLOCK
    //------------------------------------------------------------------------//
    // Calculate the interlock condition:                                     //
    //------------------------------------------------------------------------//
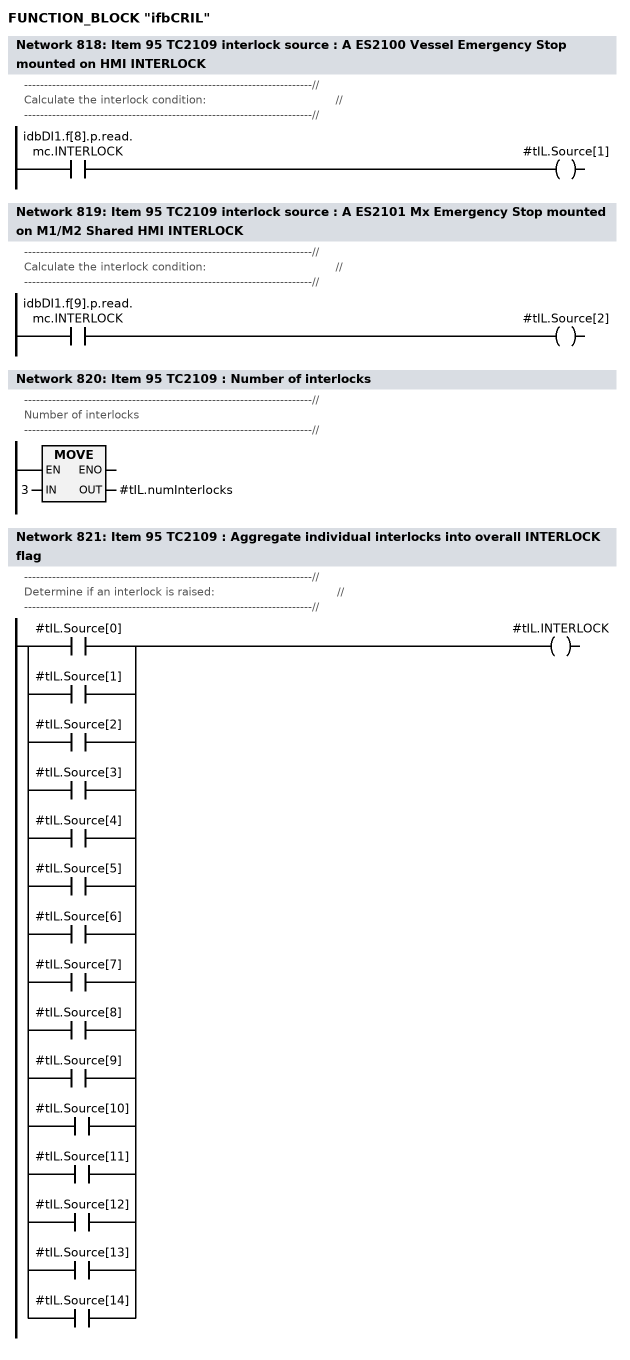
    A idbDI1.f[8].p.read.mc.INTERLOCK;
    = #tIL.Source[1];

NETWORK
TITLE = Item 95 TC2109 interlock source : A ES2101 Mx Emergency Stop mounted on M1/M2 Shared HMI INTERLOCK
    //------------------------------------------------------------------------//
    // Calculate the interlock condition:                                     //
    //------------------------------------------------------------------------//
    A idbDI1.f[9].p.read.mc.INTERLOCK;
    = #tIL.Source[2];


NETWORK
TITLE = Item 95 TC2109 : Number of interlocks
    //------------------------------------------------------------------------//
    // Number of interlocks
    //------------------------------------------------------------------------//
    L 3;
    T #tIL.numInterlocks;

NETWORK
TITLE = Item 95 TC2109 : Aggregate individual interlocks into overall INTERLOCK flag
    //------------------------------------------------------------------------//
    // Determine if an interlock is raised:                                   //
    //------------------------------------------------------------------------//
    O #tIL.Source[0];
    O #tIL.Source[1];
    O #tIL.Source[2];
    O #tIL.Source[3];
    O #tIL.Source[4];
    O #tIL.Source[5];
    O #tIL.Source[6];
    O #tIL.Source[7];
    O #tIL.Source[8];
    O #tIL.Source[9];
    O #tIL.Source[10];
    O #tIL.Source[11];
    O #tIL.Source[12];
    O #tIL.Source[13];
    O #tIL.Source[14];
    = #tIL.INTERLOCK;

NETWORK
TITLE = Item 95 TC2109 : Update the instance data
    //------------------------------------------------------------------------//
    // Update the instance DB with the calculated interlock flags:            //
    //------------------------------------------------------------------------//
    CALL MOVE
    {value_type := 'Variant'}
    (   IN                   := #tIL ,
        OUT                  := #p[95]
    );

NETWORK
TITLE = Item 96 TCV1157 : MMFLx cooling water supply control valve initialise variables
    //------------------------------------------------------------------------//
    // CRITICAL INTERLOCK   CRITICAL INTERLOCK   CRITICAL INTERLOCK   CRITICA //
    // CRITICAL INTERLOCK   CRITICAL INTERLOCK   CRITICAL INTERLOCK   CRITICA //
    //                                                                        //
    // Clear the interlock flag:                                              //
    //------------------------------------------------------------------------//
    A "alwaysLow";
    = #tIL.INTERLOCK;

    //------------------------------------------------------------------------//
    // Clear all interlock values to initialise them to off:                  //
    //------------------------------------------------------------------------//
    CALL FILL_BLK
    {value_type := 'Bool', count_type := 'UInt'}
    (   IN                   := 0 ,
        COUNT                := 15 ,
        OUT                  := #tIL.Source[0]
    );


NETWORK
TITLE = Item 96 TCV1157 interlock source : AN BAV1167 Manufacturing Filtration Line Cooling Water Supply Drain Valve CLOSED   AN BAV1169 Manufacturing Filtration Line Cooling Water Return Drain Valve CLOSED
    //------------------------------------------------------------------------//
    // Calculate the interlock condition:                                     //
    //------------------------------------------------------------------------//
    AN(;
    L "idbPOS4".f[6].p.read.mc.STATE;
    L "dbCONST".BLK.POS4.STATE.CLOSED;
    ==I;
    );
AN(;
    L "idbPOS4".f[7].p.read.mc.STATE;
    L "dbCONST".BLK.POS4.STATE.CLOSED;
    ==I;
    );
    = #tIL.Source[0];

NETWORK
TITLE = Item 96 TCV1157 interlock source : A RD1101 Vessel Burst Disc ALARM
    //------------------------------------------------------------------------//
    // Calculate the interlock condition:                                     //
    //------------------------------------------------------------------------//
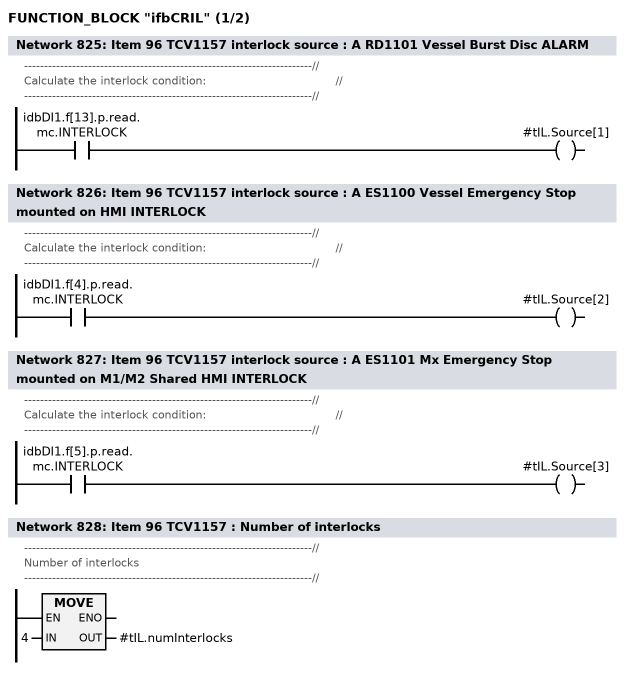
    A idbDI1.f[13].p.read.mc.INTERLOCK;
    = #tIL.Source[1];

NETWORK
TITLE = Item 96 TCV1157 interlock source : A ES1100 Vessel Emergency Stop mounted on HMI INTERLOCK
    //------------------------------------------------------------------------//
    // Calculate the interlock condition:                                     //
    //------------------------------------------------------------------------//
    A idbDI1.f[4].p.read.mc.INTERLOCK;
    = #tIL.Source[2];

NETWORK
TITLE = Item 96 TCV1157 interlock source : A ES1101 Mx Emergency Stop mounted on M1/M2 Shared HMI INTERLOCK
    //------------------------------------------------------------------------//
    // Calculate the interlock condition:                                     //
    //------------------------------------------------------------------------//
    A idbDI1.f[5].p.read.mc.INTERLOCK;
    = #tIL.Source[3];


NETWORK
TITLE = Item 96 TCV1157 : Number of interlocks
    //------------------------------------------------------------------------//
    // Number of interlocks
    //------------------------------------------------------------------------//
    L 4;
    T #tIL.numInterlocks;

NETWORK
TITLE = Item 96 TCV1157 : Aggregate individual interlocks into overall INTERLOCK flag
    //------------------------------------------------------------------------//
    // Determine if an interlock is raised:                                   //
    //------------------------------------------------------------------------//
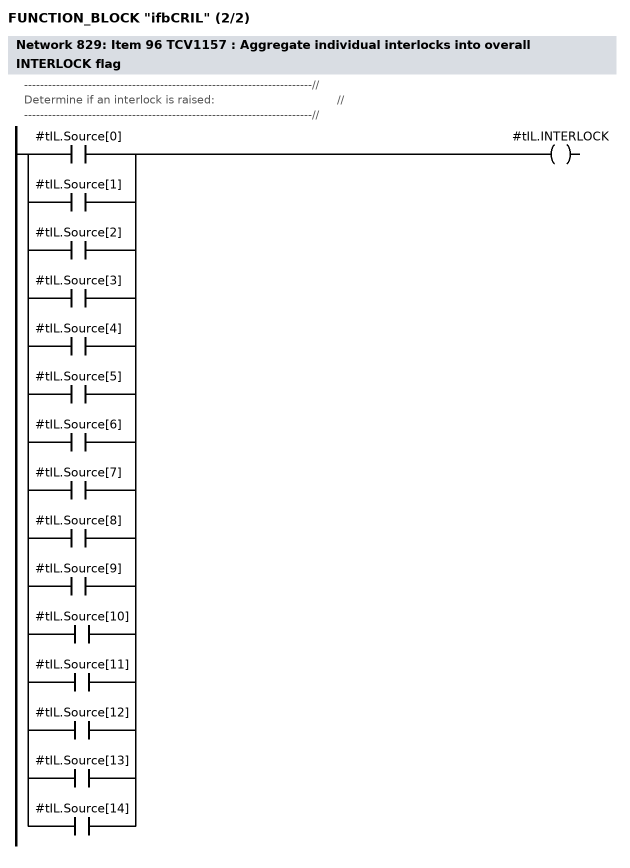
    O #tIL.Source[0];
    O #tIL.Source[1];
    O #tIL.Source[2];
    O #tIL.Source[3];
    O #tIL.Source[4];
    O #tIL.Source[5];
    O #tIL.Source[6];
    O #tIL.Source[7];
    O #tIL.Source[8];
    O #tIL.Source[9];
    O #tIL.Source[10];
    O #tIL.Source[11];
    O #tIL.Source[12];
    O #tIL.Source[13];
    O #tIL.Source[14];
    = #tIL.INTERLOCK;

NETWORK
TITLE = Item 96 TCV1157 : Update the instance data
    //------------------------------------------------------------------------//
    // Update the instance DB with the calculated interlock flags:            //
    //------------------------------------------------------------------------//
    CALL MOVE
    {value_type := 'Variant'}
    (   IN                   := #tIL ,
        OUT                  := #p[96]
    );

NETWORK
TITLE = Item 97 TCV2157 : MMFLx cooling water supply control valve initialise variables
    //------------------------------------------------------------------------//
    // CRITICAL INTERLOCK   CRITICAL INTERLOCK   CRITICAL INTERLOCK   CRITICA //
    // CRITICAL INTERLOCK   CRITICAL INTERLOCK   CRITICAL INTERLOCK   CRITICA //
    //                                                                        //
    // Clear the interlock flag:                                              //
    //------------------------------------------------------------------------//
    A "alwaysLow";
    = #tIL.INTERLOCK;

    //------------------------------------------------------------------------//
    // Clear all interlock values to initialise them to off:                  //
    //------------------------------------------------------------------------//
    CALL FILL_BLK
    {value_type := 'Bool', count_type := 'UInt'}
    (   IN                   := 0 ,
        COUNT                := 15 ,
        OUT                  := #tIL.Source[0]
    );


NETWORK
TITLE = Item 97 TCV2157 interlock source : AN BAV2167 Manufacturing Filtration Line Cooling Water Supply Drain Valve CLOSED   AN BAV2169 Manufacturing Filtration Line Cooling Water Return Drain Valve CLOSED
    //------------------------------------------------------------------------//
    // Calculate the interlock condition:                                     //
    //------------------------------------------------------------------------//
    AN(;
    L "idbPOS4".f[14].p.read.mc.STATE;
    L "dbCONST".BLK.POS4.STATE.CLOSED;
    ==I;
    );
AN(;
    L "idbPOS4".f[15].p.read.mc.STATE;
    L "dbCONST".BLK.POS4.STATE.CLOSED;
    ==I;
    );
    = #tIL.Source[0];

NETWORK
TITLE = Item 97 TCV2157 interlock source : A RD2101 Vessel Burst Disc ALARM
    //------------------------------------------------------------------------//
    // Calculate the interlock condition:                                     //
    //------------------------------------------------------------------------//
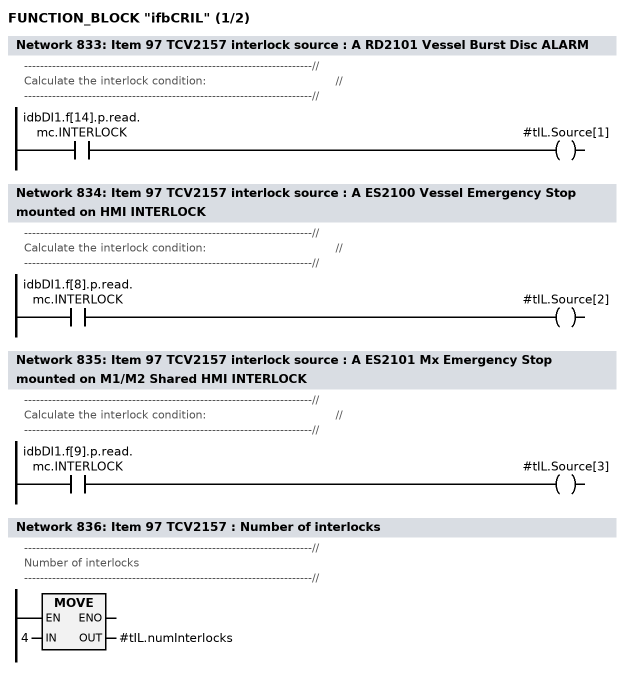
    A idbDI1.f[14].p.read.mc.INTERLOCK;
    = #tIL.Source[1];

NETWORK
TITLE = Item 97 TCV2157 interlock source : A ES2100 Vessel Emergency Stop mounted on HMI INTERLOCK
    //------------------------------------------------------------------------//
    // Calculate the interlock condition:                                     //
    //------------------------------------------------------------------------//
    A idbDI1.f[8].p.read.mc.INTERLOCK;
    = #tIL.Source[2];

NETWORK
TITLE = Item 97 TCV2157 interlock source : A ES2101 Mx Emergency Stop mounted on M1/M2 Shared HMI INTERLOCK
    //------------------------------------------------------------------------//
    // Calculate the interlock condition:                                     //
    //------------------------------------------------------------------------//
    A idbDI1.f[9].p.read.mc.INTERLOCK;
    = #tIL.Source[3];


NETWORK
TITLE = Item 97 TCV2157 : Number of interlocks
    //------------------------------------------------------------------------//
    // Number of interlocks
    //------------------------------------------------------------------------//
    L 4;
    T #tIL.numInterlocks;

NETWORK
TITLE = Item 97 TCV2157 : Aggregate individual interlocks into overall INTERLOCK flag
    //------------------------------------------------------------------------//
    // Determine if an interlock is raised:                                   //
    //------------------------------------------------------------------------//
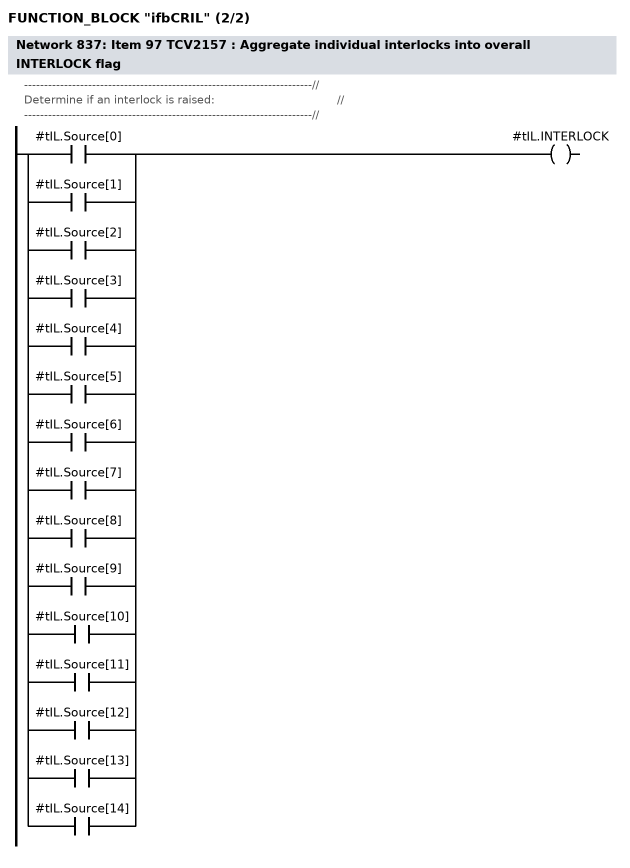
    O #tIL.Source[0];
    O #tIL.Source[1];
    O #tIL.Source[2];
    O #tIL.Source[3];
    O #tIL.Source[4];
    O #tIL.Source[5];
    O #tIL.Source[6];
    O #tIL.Source[7];
    O #tIL.Source[8];
    O #tIL.Source[9];
    O #tIL.Source[10];
    O #tIL.Source[11];
    O #tIL.Source[12];
    O #tIL.Source[13];
    O #tIL.Source[14];
    = #tIL.INTERLOCK;

NETWORK
TITLE = Item 97 TCV2157 : Update the instance data
    //------------------------------------------------------------------------//
    // Update the instance DB with the calculated interlock flags:            //
    //------------------------------------------------------------------------//
    CALL MOVE
    {value_type := 'Variant'}
    (   IN                   := #tIL ,
        OUT                  := #p[97]
    );

NETWORK
TITLE = Item 98 VP1000 : MX Vacuum Pump 1 initialise variables
    //------------------------------------------------------------------------//
    // CRITICAL INTERLOCK   CRITICAL INTERLOCK   CRITICAL INTERLOCK   CRITICA //
    // CRITICAL INTERLOCK   CRITICAL INTERLOCK   CRITICAL INTERLOCK   CRITICA //
    //                                                                        //
    // Clear the interlock flag:                                              //
    //------------------------------------------------------------------------//
    A "alwaysLow";
    = #tIL.INTERLOCK;

    //------------------------------------------------------------------------//
    // Clear all interlock values to initialise them to off:                  //
    //------------------------------------------------------------------------//
    CALL FILL_BLK
    {value_type := 'Bool', count_type := 'UInt'}
    (   IN                   := 0 ,
        COUNT                := 15 ,
        OUT                  := #tIL.Source[0]
    );


NETWORK
TITLE = Item 98 VP1000 interlock source : A ES1100 M1 Vessel Emergency Stop mounted on HMI INTERLOCK
    //------------------------------------------------------------------------//
    // Calculate the interlock condition:                                     //
    //------------------------------------------------------------------------//
    A idbDI1.f[4].p.read.mc.INTERLOCK;
    = #tIL.Source[0];

NETWORK
TITLE = Item 98 VP1000 interlock source : A ES1101 M1 Emergency Stop mounted on M1/M2 Shared HMI INTERLOCK
    //------------------------------------------------------------------------//
    // Calculate the interlock condition:                                     //
    //------------------------------------------------------------------------//
